// NeuroPLC — Auto-generated IEC 61131-3 SCL
// Graph: kan | Target: S71200Backend
// Work memory: 75KB | LUT points: 15
// Nodes: 11 | Ops: {'matmul': 3, 'standard_act': 2, 'bspline_lut': 2, 'add': 2, 'softmax': 1, 'argmax': 1}


DATA_BLOCK "NeuroPLC_Weights"
{ S7_Optimized_Access := 'FALSE' }
VERSION : 0.1
NON_RETAIN
   STRUCT

   // BsplineLUT 'l0_bspline': grid(15 pts) + table(16×28×15)
   w0 : ARRAY[0..14] OF REAL :=
[-3.0000000, -2.5714286, -2.1428571, -1.7142857, -1.2857143, -0.8571429, -0.4285714, 0.0
    0.4285714, 0.8571429, 1.2857143, 1.7142857, 2.1428571, 2.5714286, 3.0000000];
   w1 : ARRAY[0..6719] OF REAL :=
[-0.0537614, -0.0501507, -0.0466009, -0.0431086, -0.0396707, -0.0362841, -0.0329455, -0.0296518
    -0.0263998, -0.0231863, -0.0200081, -0.0168621, -0.0137450, -0.0106537, -0.0075850, 0.0036137
    0.0087966, 0.0140219, 0.0192753, 0.0245424, 0.0298091, 0.0350611, 0.0402840, 0.0454636
    0.0505857, 0.0556359, 0.0606001, 0.0654638, 0.0702129, 0.0748330, 0.0177914, 0.0204340
    0.0230393, 0.0256087, 0.0281433, 0.0306442, 0.0331128, 0.0355502, 0.0379576, 0.0403361
    0.0426870, 0.0450116, 0.0473109, 0.0495862, 0.0518386, 0.0911694, 0.0932300, 0.0951918
    0.0970447, 0.0987788, 0.1003839, 0.1018500, 0.1031669, 0.1043247, 0.1053133, 0.1061226
    0.1067426, 0.1071632, 0.1073743, 0.1073658, 0.1621530, 0.1624265, 0.1625151, 0.1624206
    0.1621450, 0.1616900, 0.1610576, 0.1602496, 0.1592678, 0.1581141, 0.1567904, 0.1552985
    0.1536403, 0.1518177, 0.1498324, 0.0235894, 0.0199670, 0.0162926, 0.0125813, 0.0088480
    0.0051075, 0.0013748, -0.0023352, -0.0060075, -0.0096273, -0.0131797, -0.0166496, -0.0200223
    -0.0232827, -0.0264160, 0.0037645, 0.0049106, 0.0061689, 0.0075391, 0.0090207, 0.0106134
    0.0123167, 0.0141303, 0.0160538, 0.0180869, 0.0202291, 0.0224800, 0.0248393, 0.0273066
    0.0298814, 0.1595527, 0.1622552, 0.1649406, 0.1675934, 0.1701985, 0.1727402, 0.1752033
    0.1775724, 0.1798320, 0.1819669, 0.1839615, 0.1858006, 0.1874687, 0.1889505, 0.1902305
    0.0697959, 0.0692244, 0.0685901, 0.0679135, 0.0672150, 0.0665149, 0.0658336, 0.0651916
    0.0646091, 0.0641067, 0.0637047, 0.0634234, 0.0632833, 0.0633048, 0.0635083, 0.0889156
    0.0916844, 0.0943388, 0.0968816, 0.0993158, 0.1016441, 0.1038697, 0.1059952, 0.1080237
    0.1099581, 0.1118012, 0.1135559, 0.1152252, 0.1168119, 0.1183189, -0.0411367, -0.0345732
    -0.0279382, -0.0212556, -0.0145492, -0.0078430, -0.0011607, 0.0054737, 0.0120364, 0.0185035
    0.0248511, 0.0310554, 0.0370926, 0.0429386, 0.0485698, 0.1426231, 0.1415560, 0.1405476
    0.1395973, 0.1387044, 0.1378686, 0.1370891, 0.1363655, 0.1356970, 0.1350832, 0.1345235
    0.1340173, 0.1335640, 0.1331631, 0.1328139, 0.2510517, 0.2566622, 0.2620918, 0.2673131
    0.2722991, 0.2770230, 0.2814575, 0.2855757, 0.2893504, 0.2927547, 0.2957615, 0.2983437
    0.3004743, 0.3021264, 0.3032727, 0.0229299, 0.0200585, 0.0170953, 0.0140589, 0.0109677
    0.0078400, 0.0046945, 0.0015496, -0.0015764, -0.0046649, -0.0076974, -0.0106555, -0.0135208
    -0.0162748, -0.0188990, 0.0368656, 0.0374461, 0.0380069, 0.0385353, 0.0390182, 0.0394428
    0.0397962, 0.0400654, 0.0402376, 0.0402999, 0.0402393, 0.0400429, 0.0396979, 0.0391914
    0.0385103, 0.2372042, 0.2373395, 0.2373046, 0.2371029, 0.2367378, 0.2362127, 0.2355310
    0.2346960, 0.2337111, 0.2325798, 0.2313054, 0.2298912, 0.2283408, 0.2266575, 0.2248445
    0.1274217, 0.1323916, 0.1373182, 0.1421699, 0.1469152, 0.1515225, 0.1559602, 0.1601968
    0.1642006, 0.1679402, 0.1713839, 0.1745002, 0.1772575, 0.1796242, 0.1815687, 0.0097799
    0.0143171, 0.0189285, 0.0236177, 0.0283886, 0.0332447, 0.0381899, 0.0432280, 0.0483625
    0.0535974, 0.0589362, 0.0643828, 0.0699409, 0.0756142, 0.0814065, 0.0746824, 0.0808143
    0.0870039, 0.0932227, 0.0994422, 0.1056337, 0.1117689, 0.1178190, 0.1237556, 0.1295501
    0.1351739, 0.1405987, 0.1457956, 0.1507363, 0.1553921, 0.1577364, 0.1559705, 0.1542206
    0.1524857, 0.1507643, 0.1490552, 0.1473571, 0.1456687, 0.1439888, 0.1423160, 0.1406490
    0.1389866, 0.1373274, 0.1356702, 0.1340137, 0.0440495, 0.0446013, 0.0452923, 0.0461173
    0.0470712, 0.0481487, 0.0493447, 0.0506540, 0.0520714, 0.0535917, 0.0552098, 0.0569205
    0.0587186, 0.0605990, 0.0625563, 0.1515065, 0.1420245, 0.1325012, 0.1229551, 0.1134045
    0.1038679, 0.0943635, 0.0849099, 0.0755254, 0.0662283, 0.0570372, 0.0479702, 0.0390460
    0.0302827, 0.0216989, 0.2110309, 0.2063019, 0.2015673, 0.1968229, 0.1920643, 0.1872871
    0.1824870, 0.1776595, 0.1728004, 0.1679052, 0.1629696, 0.1579892, 0.1529597, 0.1478766
    0.1427357, 0.1167147, 0.1155411, 0.1143786, 0.1132194, 0.1120559, 0.1108802, 0.1096847
    0.1084617, 0.1072033, 0.1059019, 0.1045497, 0.1031391, 0.1016622, 0.1001114, 0.0984789
    0.0612643, 0.0576810, 0.0542433, 0.0509556, 0.0478225, 0.0448487, 0.0420387, 0.0393971
    0.0369285, 0.0346374, 0.0325284, 0.0306060, 0.0288750, 0.0273397, 0.0260049, 0.0478268
    0.0498810, 0.0521120, 0.0545034, 0.0570387, 0.0597016, 0.0624757, 0.0653444, 0.0682915
    0.0713005, 0.0743550, 0.0774385, 0.0805347, 0.0836271, 0.0866994, 0.1196649, 0.1201896
    0.1209498, 0.1219383, 0.1231481, 0.1245723, 0.1262036, 0.1280351, 0.1300597, 0.1322704
    0.1346600, 0.1372216, 0.1399481, 0.1428323, 0.1458673, 0.1314654, 0.1267358, 0.1220911
    0.1175243, 0.1130283, 0.1085961, 0.1042207, 0.0998949, 0.0956117, 0.0913640, 0.0871449
    0.0829471, 0.0787638, 0.0745878, 0.0704120, 0.1482306, 0.1482909, 0.1482174, 0.1480233
    0.1477216, 0.1473256, 0.1468484, 0.1463031, 0.1457029, 0.1450608, 0.1443900, 0.1437037
    0.1430150, 0.1423371, 0.1416830, 0.0909267, 0.0942033, 0.0974144, 0.1005591, 0.1036367
    0.1066464, 0.1095874, 0.1124590, 0.1152604, 0.1179907, 0.1206493, 0.1232354, 0.1257481
    0.1281867, 0.1305504, 0.0411825, 0.0473991, 0.0535137, 0.0595173, 0.0654007, 0.0711547
    0.0767702, 0.0822381, 0.0875490, 0.0926940, 0.0976638, 0.1024494, 0.1070414, 0.1114309
    0.1156085, -0.1064937, -0.1066310, -0.1065970, -0.1063968, -0.1060358, -0.1055195, -0.1048531
    -0.1040420, -0.1030916, -0.1020073, -0.1007942, -0.0994579, -0.0980037, -0.0964369, -0.0947629
    0.1427321, 0.1493539, 0.1559923, 0.1626289, 0.1692458, 0.1758247, 0.1823476, 0.1887961
    0.1951523, 0.2013978, 0.2075146, 0.2134846, 0.2192896, 0.2249114, 0.2303318, 0.0604217
    0.0622943, 0.0641302, 0.0659233, 0.0676677, 0.0693572, 0.0709857, 0.0725473, 0.0740358
    0.0754452, 0.0767694, 0.0780024, 0.0791381, 0.0801705, 0.0810934, 0.1634620, 0.1628231
    0.1620056, 0.1610041, 0.1598133, 0.1584279, 0.1568425, 0.1550518, 0.1530505, 0.1508332
    0.1483946, 0.1457293, 0.1428322, 0.1396977, 0.1363206, 0.0563154, 0.0518884, 0.0473023
    0.0425774, 0.0377339, 0.0327920, 0.0277721, 0.0226943, 0.0175790, 0.0124463, 0.0073165
    0.0022098, -0.0028535, -0.0078531, -0.0127688, 0.0945771, 0.0939802, 0.0934194, 0.0929126
    0.0924782, 0.0921343, 0.0918991, 0.0917908, 0.0918276, 0.0920277, 0.0924092, 0.0929903
    0.0937893, 0.0948243, 0.0961135, 0.1597103, 0.1591299, 0.1584730, 0.1577443, 0.1569484
    0.1560901, 0.1551740, 0.1542049, 0.1531873, 0.1521261, 0.1510259, 0.1498914, 0.1487273
    0.1475383, 0.1463290, 0.1615033, 0.1660341, 0.1703599, 0.1744726, 0.1783642, 0.1820267
    0.1854521, 0.1886325, 0.1915598, 0.1942261, 0.1966232, 0.1987434, 0.2005784, 0.2021204
    0.2033613, 0.0735570, 0.0658352, 0.0581088, 0.0503981, 0.0427235, 0.0351053, 0.0275639
    0.0201196, 0.0127927, 0.0056037, -0.0014271, -0.0082794, -0.0149328, -0.0213670, -0.0275615
    0.1822264, 0.1774475, 0.1726047, 0.1676911, 0.1626996, 0.1576232, 0.1524548, 0.1471874
    0.1418141, 0.1363277, 0.1307212, 0.1249876, 0.1191199, 0.1131109, 0.1069538, 0.1921862
    0.1893261, 0.1864184, 0.1834680, 0.1804803, 0.1774603, 0.1744133, 0.1713443, 0.1682584
    0.1651610, 0.1620570, 0.1589516, 0.1558501, 0.1527575, 0.1496790, -0.0632336, -0.0648101
    -0.0662504, -0.0675372, -0.0686534, -0.0695816, -0.0703045, -0.0708049, -0.0710656, -0.0710692
    -0.0707984, -0.0702362, -0.0693650, -0.0681678, -0.0666272, 0.1172287, 0.1131316, 0.1088304
    0.1043208, 0.0995984, 0.0946590, 0.0894981, 0.0841114, 0.0784947, 0.0726435, 0.0665536
    0.0602206, 0.0536403, 0.0468081, 0.0397199, 0.1591443, 0.1524481, 0.1457851, 0.1391899
    0.1326966, 0.1263399, 0.1201540, 0.1141734, 0.1084325, 0.1029658, 0.0978075, 0.0929922
    0.0885542, 0.0845280, 0.0809479, -0.0802141, -0.0751070, -0.0699127, -0.0646468, -0.0593249
    -0.0539626, -0.0485752, -0.0431786, -0.0377880, -0.0324192, -0.0270877, -0.0218090, -0.0165986
    -0.0114722, -0.0064453, 0.0824098, 0.0763993, 0.0705333, 0.0648235, 0.0592816, 0.0539193
    0.0487485, 0.0437808, 0.0390279, 0.0345016, 0.0302137, 0.0261759, 0.0223999, 0.0188974
    0.0156802, 0.1799797, 0.1784663, 0.1767808, 0.1749217, 0.1728874, 0.1706764, 0.1682869
    0.1657176, 0.1629667, 0.1600327, 0.1569141, 0.1536092, 0.1501164, 0.1464343, 0.1425611
    -0.0496284, -0.0452828, -0.0409373, -0.0365933, -0.0322526, -0.0279167, -0.0235873, -0.0192659
    -0.0149543, -0.0106539, -0.0063663, -0.0020933, 0.0021636, 0.0064028, 0.0106226, 0.0450445
    0.0502692, 0.0554434, 0.0605487, 0.0655669, 0.0704798, 0.0752689, 0.0799160, 0.0844028
    0.0887111, 0.0928225, 0.0967188, 0.1003817, 0.1037928, 0.1069339, -0.0646169, -0.0560196
    -0.0472858, -0.0384308, -0.0294704, -0.0204202, -0.0112958, -0.0021127, 0.0071135, 0.0163671
    0.0256325, 0.0348942, 0.0441365, 0.0533439, 0.0625006, 0.0364423, 0.0390047, 0.0413258
    0.0434204, 0.0453037, 0.0469907, 0.0484963, 0.0498356, 0.0510236, 0.0520753, 0.0530057
    0.0538298, 0.0545627, 0.0552193, 0.0558146, 0.1494066, 0.1454436, 0.1415708, 0.1377844
    0.1340804, 0.1304549, 0.1269041, 0.1234239, 0.1200105, 0.1166601, 0.1133685, 0.1101320
    0.1069467, 0.1038086, 0.1007139, -0.0151529, -0.0096418, -0.0041800, 0.0012205, 0.0065474
    0.0117887, 0.0169322, 0.0219657, 0.0268772, 0.0316544, 0.0362853, 0.0407577, 0.0450594
    0.0491783, 0.0531024, 0.0760455, 0.0828511, 0.0895923, 0.0962519, 0.1028127, 0.1092577
    0.1155697, 0.1217317, 0.1277264, 0.1335369, 0.1391458, 0.1445363, 0.1496910, 0.1545929
    0.1592250, -0.0199655, -0.0125562, -0.0050469, 0.0025438, 0.0101974, 0.0178952, 0.0256188
    0.0333496, 0.0410690, 0.0487583, 0.0563991, 0.0639728, 0.0714608, 0.0788445, 0.0861054
    -0.0196776, -0.0178736, -0.0159748, -0.0139721, -0.0118560, -0.0096175, -0.0072471, -0.0047358
    -0.0020741, 0.0007470, 0.0037369, 0.0069048, 0.0102600, 0.0138117, 0.0175692, 0.0124894
    0.0173022, 0.0219949, 0.0265723, 0.0310388, 0.0353992, 0.0396580, 0.0438199, 0.0478895
    0.0518714, 0.0557702, 0.0595906, 0.0633373, 0.0670147, 0.0706276, 0.0248611, 0.0284164
    0.0320837, 0.0358641, 0.0397584, 0.0437678, 0.0478931, 0.0521354, 0.0564957, 0.0609750
    0.0655743, 0.0702945, 0.0751367, 0.0801018, 0.0851909, 0.1490314, 0.1533812, 0.1576221
    0.1617333, 0.1656937, 0.1694824, 0.1730786, 0.1764612, 0.1796093, 0.1825020, 0.1851182
    0.1874372, 0.1894379, 0.1910994, 0.1924008, 0.0541098, 0.0578787, 0.0616169, 0.0652991
    0.0689002, 0.0723947, 0.0757576, 0.0789636, 0.0819875, 0.0848040, 0.0873880, 0.0897141
    0.0917573, 0.0934922, 0.0948936, 0.0617447, 0.0675283, 0.0733681, 0.0792395, 0.0851180
    0.0909790, 0.0967979, 0.1025502, 0.1082113, 0.1137566, 0.1191614, 0.1244014, 0.1294519
    0.1342882, 0.1388859, -0.0461591, -0.0453256, -0.0443076, -0.0431073, -0.0417270, -0.0401691
    -0.0384360, -0.0365298, -0.0344530, -0.0322079, -0.0297967, -0.0272219, -0.0244857, -0.0215905
    -0.0185385, 0.0292693, 0.0302004, 0.0311640, 0.0321651, 0.0332088, 0.0343000, 0.0354438
    0.0366453, 0.0379094, 0.0392413, 0.0406458, 0.0421281, 0.0436931, 0.0453460, 0.0470917
    0.1551978, 0.1594762, 0.1635234, 0.1673317, 0.1708932, 0.1742002, 0.1772451, 0.1800199
    0.1825169, 0.1847285, 0.1866468, 0.1882641, 0.1895726, 0.1905645, 0.1912322, -0.0022298
    0.0015482, 0.0054057, 0.0093347, 0.0133276, 0.0173766, 0.0214738, 0.0256116, 0.0297821
    0.0339775, 0.0381901, 0.0424120, 0.0466356, 0.0508530, 0.0550565, 0.0832689, 0.0901474
    0.0970738, 0.1040439, 0.1110534, 0.1180982, 0.1251741, 0.1322769, 0.1394024, 0.1465464
    0.1537047, 0.1608732, 0.1680476, 0.1752237, 0.1823975, 0.0709989, 0.0702285, 0.0696263
    0.0691951, 0.0689377, 0.0688570, 0.0689556, 0.0692364, 0.0697023, 0.0703559, 0.0712001
    0.0722376, 0.0734714, 0.0749041, 0.0765386, 0.0713218, 0.0738626, 0.0762200, 0.0783959
    0.0803921, 0.0822106, 0.0838531, 0.0853217, 0.0866181, 0.0877443, 0.0887021, 0.0894935
    0.0901202, 0.0905842, 0.0908874, 0.1406779, 0.1441289, 0.1474667, 0.1506924, 0.1538070
    0.1568115, 0.1597070, 0.1624945, 0.1651749, 0.1677495, 0.1702191, 0.1725848, 0.1748478
    0.1770088, 0.1790691, 0.0130739, 0.0090535, 0.0049917, 0.0009004, -0.0032088, -0.0073243
    -0.0114343, -0.0155273, -0.0195916, -0.0236154, -0.0275873, -0.0314954, -0.0353281, -0.0390738
    -0.0427207, 0.0809735, 0.0798324, 0.0785689, 0.0771792, 0.0756592, 0.0740052, 0.0722131
    0.0702792, 0.0681993, 0.0659697, 0.0635865, 0.0610456, 0.0583432, 0.0554754, 0.0524383
    0.1908756, 0.1884213, 0.1857675, 0.1829149, 0.1798646, 0.1766175, 0.1731745, 0.1695365
    0.1657044, 0.1616793, 0.1574618, 0.1530531, 0.1484540, 0.1436654, 0.1386883, -0.1181388
    -0.1128441, -0.1073974, -0.1018071, -0.0960813, -0.0902284, -0.0842566, -0.0781741, -0.0719893
    -0.0657102, -0.0593453, -0.0529027, -0.0463907, -0.0398176, -0.0331916, -0.0020498, 0.0079060
    0.0177509, 0.0274740, 0.0370644, 0.0465111, 0.0558031, 0.0649296, 0.0738794, 0.0826418
    0.0912057, 0.0995603, 0.1076945, 0.1155974, 0.1232580, -0.0007446, -0.0019150, -0.0031143
    -0.0043173, -0.0054990, -0.0066342, -0.0076977, -0.0086645, -0.0095093, -0.0102072, -0.0107328
    -0.0110612, -0.0111671, -0.0110255, -0.0106112, 0.1774268, 0.1753455, 0.1732356, 0.1710882
    0.1688946, 0.1666464, 0.1643346, 0.1619507, 0.1594860, 0.1569317, 0.1542792, 0.1515199
    0.1486450, 0.1456458, 0.1425137, 0.1379051, 0.1349382, 0.1318155, 0.1285463, 0.1251401
    0.1216064, 0.1179545, 0.1141940, 0.1103341, 0.1063845, 0.1023545, 0.0982536, 0.0940911
    0.0898766, 0.0856195, 0.0633166, 0.0493134, 0.0352768, 0.0212369, 0.0072238, -0.0067325
    -0.0206019, -0.0343543, -0.0479595, -0.0613876, -0.0746085, -0.0875920, -0.1003081, -0.1127267
    -0.1248178, 0.1183318, 0.1136023, 0.1089029, 0.1042314, 0.0995855, 0.0949629, 0.0903612
    0.0857784, 0.0812119, 0.0766596, 0.0721192, 0.0675883, 0.0630647, 0.0585461, 0.0540302
    0.1106823, 0.1041894, 0.0975902, 0.0909071, 0.0841626, 0.0773792, 0.0705792, 0.0637853
    0.0570198, 0.0503051, 0.0436638, 0.0371183, 0.0306911, 0.0244045, 0.0182812, 0.0562573
    0.0481918, 0.0400543, 0.0318683, 0.0236572, 0.0154445, 0.0072537, -0.0008917, -0.0089682
    -0.0169524, -0.0248208, -0.0325500, -0.0401163, -0.0474965, -0.0546669, 0.2219241, 0.2176533
    0.2134451, 0.2093052, 0.2052390, 0.2012524, 0.1973507, 0.1935398, 0.1898251, 0.1862123
    0.1827069, 0.1793146, 0.1760410, 0.1728917, 0.1698723, 0.3312375, 0.3261927, 0.3209868
    0.3156299, 0.3101325, 0.3045048, 0.2987574, 0.2929004, 0.2869442, 0.2808991, 0.2747756
    0.2685839, 0.2623343, 0.2560374, 0.2497033, 0.1718789, 0.1756587, 0.1793987, 0.1830900
    0.1867239, 0.1902918, 0.1937850, 0.1971947, 0.2005122, 0.2037288, 0.2068357, 0.2098243
    0.2126858, 0.2154116, 0.2179928, 0.1224311, 0.1282386, 0.1340468, 0.1398439, 0.1456182
    0.1513580, 0.1570517, 0.1626873, 0.1682533, 0.1737379, 0.1791293, 0.1844160, 0.1895860
    0.1946277, 0.1995294, 0.0492804, 0.0562029, 0.0630472, 0.0698060, 0.0764722, 0.0830386
    0.0894981, 0.0958434, 0.1020674, 0.1081630, 0.1141229, 0.1199399, 0.1256070, 0.1311170
    0.1364626, 0.1061752, 0.1096911, 0.1131474, 0.1165290, 0.1198208, 0.1230075, 0.1260742
    0.1290057, 0.1317867, 0.1344023, 0.1368373, 0.1390765, 0.1411048, 0.1429072, 0.1444684
    0.0055067, 0.0101075, 0.0148682, 0.0197738, 0.0248092, 0.0299594, 0.0352094, 0.0405440
    0.0459484, 0.0514074, 0.0569060, 0.0624292, 0.0679618, 0.0734890, 0.0789956, 0.2030336
    0.2064162, 0.2097383, 0.2129931, 0.2161737, 0.2192730, 0.2222843, 0.2252005, 0.2280147
    0.2307200, 0.2333094, 0.2357761, 0.2381131, 0.2403134, 0.2423701, 0.0904342, 0.0915991
    0.0928258, 0.0941062, 0.0954321, 0.0967953, 0.0981878, 0.0996012, 0.1010275, 0.1024584
    0.1038859, 0.1053016, 0.1066976, 0.1080655, 0.1093972, 0.1280624, 0.1273501, 0.1266980
    0.1261149, 0.1256098, 0.1251912, 0.1248681, 0.1246492, 0.1245433, 0.1245592, 0.1247057
    0.1249917, 0.1254258, 0.1260169, 0.1267738, 0.1299709, 0.1307576, 0.1315505, 0.1323500
    0.1331564, 0.1339704, 0.1347923, 0.1356225, 0.1364616, 0.1373100, 0.1381681, 0.1390364
    0.1399154, 0.1408054, 0.1417070, 0.1533135, 0.1507089, 0.1480348, 0.1452944, 0.1424904
    0.1396261, 0.1367043, 0.1337281, 0.1307005, 0.1276246, 0.1245032, 0.1213395, 0.1181364
    0.1148970, 0.1116242, 0.0754236, 0.0751954, 0.0749772, 0.0747602, 0.0745356, 0.0742946
    0.0740284, 0.0737282, 0.0733853, 0.0729909, 0.0725361, 0.0720122, 0.0714104, 0.0707219
    0.0699379, 0.2758769, 0.2724863, 0.2687611, 0.2647197, 0.2603807, 0.2557624, 0.2508835
    0.2457622, 0.2404172, 0.2348669, 0.2291298, 0.2232242, 0.2171688, 0.2109820, 0.2046822
    0.0770989, 0.0772505, 0.0775468, 0.0779858, 0.0785653, 0.0792835, 0.0801382, 0.0811273
    0.0822489, 0.0835009, 0.0848812, 0.0863879, 0.0880188, 0.0897719, 0.0916453, 0.1377456
    0.1380898, 0.1384590, 0.1388540, 0.1392763, 0.1397269, 0.1402069, 0.1407176, 0.1412600
    0.1418354, 0.1424448, 0.1430894, 0.1437705, 0.1444890, 0.1452463, 0.0905914, 0.0893503
    0.0881403, 0.0869641, 0.0858247, 0.0847249, 0.0836674, 0.0826551, 0.0816908, 0.0807774
    0.0799175, 0.0791142, 0.0783702, 0.0776883, 0.0770713, 0.0768078, 0.0747090, 0.0725560
    0.0703614, 0.0681377, 0.0658974, 0.0636532, 0.0614176, 0.0592031, 0.0570223, 0.0548878
    0.0528120, 0.0508076, 0.0488871, 0.0470630, 0.0018665, 0.0055140, 0.0092878, 0.0131758
    0.0171657, 0.0212453, 0.0254025, 0.0296251, 0.0339007, 0.0382174, 0.0425627, 0.0469246
    0.0512909, 0.0556493, 0.0599876, 0.1362334, 0.1320360, 0.1276240, 0.1230101, 0.1182072
    0.1132279, 0.1080852, 0.1027917, 0.0973602, 0.0918035, 0.0861343, 0.0803655, 0.0745097
    0.0685798, 0.0625885, 0.0739216, 0.0777187, 0.0816159, 0.0855995, 0.0896565, 0.0937732
    0.0979364, 0.1021327, 0.1063487, 0.1105710, 0.1147861, 0.1189809, 0.1231417, 0.1272554
    0.1313084, 0.1225641, 0.1228170, 0.1230709, 0.1233162, 0.1235429, 0.1237414, 0.1239020
    0.1240148, 0.1240701, 0.1240582, 0.1239692, 0.1237935, 0.1235212, 0.1231427, 0.1226481
    0.0764033, 0.0779041, 0.0794761, 0.0811008, 0.0827599, 0.0844351, 0.0861080, 0.0877602
    0.0893733, 0.0909290, 0.0924088, 0.0937945, 0.0950676, 0.0962098, 0.0972026, 0.1156939
    0.1193963, 0.1228430, 0.1260415, 0.1289993, 0.1317239, 0.1342227, 0.1365035, 0.1385735
    0.1404405, 0.1421117, 0.1435948, 0.1448973, 0.1460266, 0.1469904, 0.0673942, 0.0704027
    0.0733808, 0.0763299, 0.0792510, 0.0821455, 0.0850145, 0.0878592, 0.0906810, 0.0934810
    0.0962604, 0.0990204, 0.1017624, 0.1044874, 0.1071967, 0.0388152, 0.0469437, 0.0549675
    0.0628623, 0.0706043, 0.0781692, 0.0855331, 0.0926718, 0.0995613, 0.1061776, 0.1124965
    0.1184940, 0.1241459, 0.1294284, 0.1343171, 0.1772938, 0.1717090, 0.1661408, 0.1606062
    0.1551221, 0.1497055, 0.1443732, 0.1391423, 0.1340295, 0.1290519, 0.1242263, 0.1195697
    0.1150991, 0.1108312, 0.1067832, 0.1667371, 0.1745140, 0.1819698, 0.1890907, 0.1958626
    0.2022715, 0.2083035, 0.2139444, 0.2191803, 0.2239972, 0.2283811, 0.2323180, 0.2357939
    0.2387947, 0.2413065, 0.1465034, 0.1458727, 0.1451484, 0.1443270, 0.1434050, 0.1423789
    0.1412452, 0.1400004, 0.1386409, 0.1371633, 0.1355640, 0.1338395, 0.1319864, 0.1300010
    0.1278800, -0.1464676, -0.1331242, -0.1196480, -0.1060719, -0.0924292, -0.0787528, -0.0650760
    -0.0514318, -0.0378533, -0.0243737, -0.0110261, 0.0021565, 0.0151410, 0.0278942, 0.0403829
    0.0219379, 0.0184042, 0.0149580, 0.0116003, 0.0083324, 0.0051556, 0.0020711, -0.0009198
    -0.0038158, -0.0066158, -0.0093184, -0.0119225, -0.0144268, -0.0168299, -0.0191308, -0.0799424
    -0.0830510, -0.0860327, -0.0888876, -0.0916160, -0.0942182, -0.0966944, -0.0990448, -0.1012698
    -0.1033695, -0.1053442, -0.1071942, -0.1089198, -0.1105211, -0.1119984, 0.1063759, 0.1058369
    0.1052956, 0.1047466, 0.1041849, 0.1036053, 0.1030025, 0.1023714, 0.1017069, 0.1010037
    0.1002566, 0.0994605, 0.0986103, 0.0977007, 0.0967265, -0.0524474, -0.0499474, -0.0472491
    -0.0443565, -0.0412736, -0.0380045, -0.0345532, -0.0309238, -0.0271203, -0.0231467, -0.0190072
    -0.0147057, -0.0102462, -0.0056329, -0.0008698, -0.0401886, -0.0425021, -0.0449156, -0.0474036
    -0.0499410, -0.0525023, -0.0550621, -0.0575950, -0.0600758, -0.0624789, -0.0647791, -0.0669510
    -0.0689691, -0.0708082, -0.0724429, 0.0068997, 0.0025731, -0.0018010, -0.0061969, -0.0105893
    -0.0149526, -0.0192613, -0.0234899, -0.0276128, -0.0316047, -0.0354398, -0.0390929, -0.0425383
    -0.0457506, -0.0487042, 0.0460935, 0.0446672, 0.0431436, 0.0415249, 0.0398133, 0.0380112
    0.0361207, 0.0341442, 0.0320837, 0.0299417, 0.0277203, 0.0254217, 0.0230483, 0.0206022
    0.0180857, 0.0362551, 0.0359917, 0.0356584, 0.0352565, 0.0347877, 0.0342534, 0.0336551
    0.0329943, 0.0322726, 0.0314914, 0.0306522, 0.0297565, 0.0288058, 0.0278016, 0.0267454
    0.1229962, 0.1128694, 0.1027529, 0.0926827, 0.0826947, 0.0728249, 0.0631090, 0.0535829
    0.0442827, 0.0352441, 0.0265031, 0.0180955, 0.0100574, 0.0024244, -0.0047673, -0.0390921
    -0.0409484, -0.0426025, -0.0440575, -0.0453165, -0.0463824, -0.0472584, -0.0479475, -0.0484527
    -0.0487771, -0.0489238, -0.0488957, -0.0486959, -0.0483276, -0.0477937, 0.0402361, 0.0420451
    0.0438251, 0.0455756, 0.0472959, 0.0489854, 0.0506435, 0.0522696, 0.0538632, 0.0554235
    0.0569500, 0.0584422, 0.0598992, 0.0613207, 0.0627060, -0.0578378, -0.0600211, -0.0621784
    -0.0642941, -0.0663524, -0.0683375, -0.0702337, -0.0720250, -0.0736959, -0.0752304, -0.0766129
    -0.0778275, -0.0788584, -0.0796900, -0.0803063, -0.0276505, -0.0345807, -0.0413763, -0.0480331
    -0.0545471, -0.0609143, -0.0671306, -0.0731920, -0.0790944, -0.0848337, -0.0904060, -0.0958071
    -0.1010331, -0.1060798, -0.1109432, -0.0786863, -0.0790071, -0.0793080, -0.0795758, -0.0797971
    -0.0799585, -0.0800469, -0.0800488, -0.0799510, -0.0797402, -0.0794029, -0.0789260, -0.0782961
    -0.0774999, -0.0765241, 0.0213712, 0.0235205, 0.0256513, 0.0277667, 0.0298702, 0.0319649
    0.0340539, 0.0361407, 0.0382283, 0.0403200, 0.0424190, 0.0445287, 0.0466521, 0.0487925
    0.0509532, 0.0470440, 0.0409675, 0.0348353, 0.0286634, 0.0224677, 0.0162640, 0.0100684
    0.0038966, -0.0022354, -0.0083116, -0.0143163, -0.0202335, -0.0260472, -0.0317417, -0.0373009
    0.0554819, 0.0524533, 0.0493854, 0.0462786, 0.0431332, 0.0399497, 0.0367285, 0.0334701
    0.0301748, 0.0268430, 0.0234752, 0.0200718, 0.0166333, 0.0131599, 0.0096522, -0.0472854
    -0.0443733, -0.0413744, -0.0382941, -0.0351381, -0.0319120, -0.0286213, -0.0252716, -0.0218685
    -0.0184174, -0.0149240, -0.0113939, -0.0078326, -0.0042456, -0.0006386, 0.2066563, 0.1984604
    0.1899513, 0.1811467, 0.1720641, 0.1627212, 0.1531354, 0.1433243, 0.1333057, 0.1230969
    0.1127157, 0.1021795, 0.0915059, 0.0807126, 0.0698171, 0.2430425, 0.2368604, 0.2303846
    0.2236263, 0.2165967, 0.2093072, 0.2017691, 0.1939936, 0.1859921, 0.1777758, 0.1693560
    0.1607441, 0.1519513, 0.1429889, 0.1338682, -0.2294966, -0.2238292, -0.2179271, -0.2117862
    -0.2054024, -0.1987716, -0.1918898, -0.1847527, -0.1773564, -0.1696967, -0.1617694, -0.1535706
    -0.1450962, -0.1363419, -0.1273037, -0.0534835, -0.0518626, -0.0502081, -0.0485070, -0.0467464
    -0.0449133, -0.0429948, -0.0409777, -0.0388492, -0.0365964, -0.0342061, -0.0316654, -0.0289615
    -0.0260812, -0.0230116, -0.0738918, -0.0681270, -0.0624695, -0.0569120, -0.0514472, -0.0460679
    -0.0407668, -0.0355367, -0.0303702, -0.0252601, -0.0201992, -0.0151801, -0.0101956, -0.0052385
    -0.0003014, -0.1733572, -0.1706521, -0.1679701, -0.1652953, -0.1626123, -0.1599054, -0.1571589
    -0.1543573, -0.1514847, -0.1485257, -0.1454645, -0.1422856, -0.1389732, -0.1355117, -0.1318855
    -0.1211167, -0.1186958, -0.1162400, -0.1137493, -0.1112237, -0.1086634, -0.1060684, -0.1034386
    -0.1007743, -0.0980754, -0.0953419, -0.0925739, -0.0897715, -0.0869348, -0.0840637, -0.1646881
    -0.1559299, -0.1470360, -0.1380355, -0.1289572, -0.1198299, -0.1106827, -0.1015443, -0.0924438
    -0.0834100, -0.0744717, -0.0656579, -0.0569975, -0.0485193, -0.0402523, -0.0817973, -0.0730933
    -0.0642312, -0.0552295, -0.0461065, -0.0368805, -0.0275698, -0.0181927, -0.0087677, 0.0006871
    0.0101533, 0.0196125, 0.0290465, 0.0384369, 0.0477654, 0.0163655, 0.0131517, 0.0101446
    0.0073348, 0.0047129, 0.0022695, -0.0000050, -0.0021197, -0.0040842, -0.0059079, -0.0076002
    -0.0091705, -0.0106281, -0.0119826, -0.0132432, 0.1066189, 0.1081075, 0.1096451, 0.1112214
    0.1128261, 0.1144488, 0.1160794, 0.1177076, 0.1193229, 0.1209153, 0.1224743, 0.1239896
    0.1254511, 0.1268484, 0.1281711, 0.1267634, 0.1300867, 0.1334209, 0.1367561, 0.1400827
    0.1433908, 0.1466706, 0.1499123, 0.1531061, 0.1562422, 0.1593107, 0.1623020, 0.1652061
    0.1680134, 0.1707140, 0.1024532, 0.1037427, 0.1049064, 0.1059469, 0.1068673, 0.1076704
    0.1083589, 0.1089356, 0.1094036, 0.1097654, 0.1100241, 0.1101824, 0.1102432, 0.1102092
    0.1100834, 0.0440706, 0.0458766, 0.0476553, 0.0494080, 0.0511363, 0.0528416, 0.0545253
    0.0561887, 0.0578334, 0.0594607, 0.0610720, 0.0626688, 0.0642525, 0.0658246, 0.0673864
    -0.0485841, -0.0409054, -0.0330825, -0.0251116, -0.0169887, -0.0087100, -0.0002714, 0.0083308
    0.0171006, 0.0260419, 0.0351585, 0.0444545, 0.0539337, 0.0636000, 0.0734574, 0.1719400
    0.1734631, 0.1749307, 0.1763346, 0.1776664, 0.1789180, 0.1800810, 0.1811472, 0.1821083
    0.1829559, 0.1836818, 0.1842779, 0.1847356, 0.1850469, 0.1852033, 0.0836945, 0.0829144
    0.0820091, 0.0809680, 0.0797808, 0.0784369, 0.0769259, 0.0752372, 0.0733605, 0.0712852
    0.0690009, 0.0664970, 0.0637631, 0.0607888, 0.0575636, 0.0451547, 0.0443564, 0.0433699
    0.0422019, 0.0408591, 0.0393482, 0.0376759, 0.0358490, 0.0338742, 0.0317582, 0.0295077
    0.0271295, 0.0246304, 0.0220170, 0.0192960, 0.1446830, 0.1442651, 0.1438369, 0.1434112
    0.1430013, 0.1426201, 0.1422805, 0.1419956, 0.1417785, 0.1416420, 0.1415993, 0.1416632
    0.1418470, 0.1421634, 0.1426256, -0.0780212, -0.0782113, -0.0783461, -0.0784252, -0.0784484
    -0.0784154, -0.0783258, -0.0781794, -0.0779759, -0.0777149, -0.0773962, -0.0770194, -0.0765842
    -0.0760904, -0.0755376, 0.2056785, 0.2034542, 0.2009305, 0.1981261, 0.1950600, 0.1917508
    0.1882173, 0.1844784, 0.1805528, 0.1764593, 0.1722167, 0.1678438, 0.1633593, 0.1587822
    0.1541310, 0.1056817, 0.0955098, 0.0850380, 0.0743014, 0.0633348, 0.0521733, 0.0408519
    0.0294056, 0.0178693, 0.0062781, -0.0053330, -0.0169291, -0.0284751, -0.0399361, -0.0512770
    0.0299433, 0.0223843, 0.0149406, 0.0076058, 0.0003734, -0.0067630, -0.0138100, -0.0207740
    -0.0276615, -0.0344789, -0.0412327, -0.0479294, -0.0545755, -0.0611774, -0.0677417, 0.1432800
    0.1365236, 0.1298036, 0.1231296, 0.1165111, 0.1099579, 0.1034795, 0.0970856, 0.0907857
    0.0845895, 0.0785066, 0.0725466, 0.0667192, 0.0610339, 0.0555004, -0.0302912, -0.0280554
    -0.0257948, -0.0235061, -0.0211860, -0.0188312, -0.0164385, -0.0140044, -0.0115256, -0.0089990
    -0.0064211, -0.0037886, -0.0010983, 0.0016532, 0.0044692, 0.1403525, 0.1435867, 0.1466069
    0.1493943, 0.1519307, 0.1541973, 0.1561757, 0.1578473, 0.1591936, 0.1601962, 0.1608364
    0.1610958, 0.1609558, 0.1603979, 0.1594036, -0.0224080, -0.0231706, -0.0235986, -0.0236903
    -0.0234441, -0.0228584, -0.0219317, -0.0206623, -0.0190486, -0.0170891, -0.0147821, -0.0121260
    -0.0091192, -0.0057602, -0.0020472, 0.0048894, 0.0037833, 0.0026298, 0.0014329, 0.0001967
    -0.0010748, -0.0023775, -0.0037073, -0.0050602, -0.0064321, -0.0078189, -0.0092166, -0.0106211
    -0.0120284, -0.0134344, 0.1748016, 0.1674656, 0.1599554, 0.1522917, 0.1444954, 0.1365874
    0.1285885, 0.1205195, 0.1124012, 0.1042545, 0.0961002, 0.0879591, 0.0798522, 0.0718001
    0.0638238, 0.2813404, 0.2743131, 0.2670321, 0.2595086, 0.2517535, 0.2437782, 0.2355935
    0.2272108, 0.2186410, 0.2098953, 0.2009848, 0.1919205, 0.1827137, 0.1733754, 0.1639168
    -0.1227151, -0.1167440, -0.1105694, -0.1042075, -0.0976747, -0.0909872, -0.0841613, -0.0772134
    -0.0701597, -0.0630166, -0.0558003, -0.0485272, -0.0412136, -0.0338758, -0.0265300, 0.0716502
    0.0740325, 0.0763472, 0.0785967, 0.0807833, 0.0829093, 0.0849771, 0.0869889, 0.0889471
    0.0908540, 0.0927120, 0.0945233, 0.0962903, 0.0980153, 0.0997006, 0.1102683, 0.1225627
    0.1347638, 0.1468584, 0.1588335, 0.1706758, 0.1823722, 0.1939096, 0.2052749, 0.2164549
    0.2274364, 0.2382064, 0.2487517, 0.2590591, 0.2691154, 0.2098262, 0.2144697, 0.2187104
    0.2225624, 0.2260398, 0.2291567, 0.2319272, 0.2343654, 0.2364854, 0.2383013, 0.2398272
    0.2410773, 0.2420656, 0.2428063, 0.2433134, 0.1236384, 0.1234346, 0.1231693, 0.1228465
    0.1224701, 0.1220440, 0.1215722, 0.1210586, 0.1205071, 0.1199218, 0.1193064, 0.1186650
    0.1180016, 0.1173200, 0.1166241, -0.0358423, -0.0302241, -0.0246765, -0.0192003, -0.0137963
    -0.0084654, -0.0032083, 0.0019742, 0.0070812, 0.0121121, 0.0170660, 0.0219421, 0.0267396
    0.0314578, 0.0360958, -0.0184696, -0.0128896, -0.0074545, -0.0021679, 0.0029665, 0.0079452
    0.0127643, 0.0174204, 0.0219097, 0.0262287, 0.0303736, 0.0343408, 0.0381267, 0.0417277
    0.0451400, -0.1589818, -0.1530462, -0.1471289, -0.1412169, -0.1352974, -0.1293573, -0.1233838
    -0.1173639, -0.1112847, -0.1051332, -0.0988965, -0.0925616, -0.0861157, -0.0795457, -0.0728388
    -0.0915808, -0.0858980, -0.0802137, -0.0745331, -0.0688611, -0.0632027, -0.0575628, -0.0519466
    -0.0463591, -0.0408051, -0.0352897, -0.0298179, -0.0243948, -0.0190252, -0.0137143, -0.0835398
    -0.0728436, -0.0621097, -0.0513475, -0.0405668, -0.0297773, -0.0189886, -0.0082104, 0.0025477
    0.0132760, 0.0239648, 0.0346044, 0.0451853, 0.0556977, 0.0661319, -0.0592816, -0.0595268
    -0.0600139, -0.0607121, -0.0615909, -0.0626199, -0.0637683, -0.0650056, -0.0663012, -0.0676246
    -0.0689452, -0.0702323, -0.0714555, -0.0725841, -0.0735876, 0.0978256, 0.0979407, 0.0979876
    0.0979614, 0.0978575, 0.0976711, 0.0973975, 0.0970319, 0.0965695, 0.0960057, 0.0953356
    0.0945545, 0.0936577, 0.0926404, 0.0914979, -0.1088112, -0.1062184, -0.1035894, -0.1009293
    -0.0982433, -0.0955364, -0.0928137, -0.0900805, -0.0873417, -0.0846026, -0.0818682, -0.0791436
    -0.0764340, -0.0737444, -0.0710801, 0.0581553, 0.0553071, 0.0523084, 0.0491769, 0.0459304
    0.0425867, 0.0391635, 0.0356786, 0.0321498, 0.0285947, 0.0250312, 0.0214770, 0.0179500
    0.0144677, 0.0110481, -0.0312003, -0.0265061, -0.0215812, -0.0164328, -0.0110683, -0.0054952
    0.0002792, 0.0062476, 0.0124024, 0.0187363, 0.0252420, 0.0319121, 0.0387391, 0.0457157
    0.0528345, 0.0662310, 0.0672577, 0.0681709, 0.0689749, 0.0696742, 0.0702732, 0.0707762
    0.0711877, 0.0715121, 0.0717537, 0.0719170, 0.0720064, 0.0720262, 0.0719809, 0.0718749
    -0.0591723, -0.0535568, -0.0479641, -0.0424035, -0.0368841, -0.0314154, -0.0260063, -0.0206662
    -0.0154042, -0.0102296, -0.0051516, -0.0001794, 0.0046778, 0.0094108, 0.0140103, 0.1534036
    0.1555018, 0.1573710, 0.1590074, 0.1604071, 0.1615662, 0.1624808, 0.1631471, 0.1635612
    0.1637191, 0.1636170, 0.1632512, 0.1626176, 0.1617124, 0.1605317, -0.0163877, -0.0142709
    -0.0121985, -0.0101703, -0.0081860, -0.0062452, -0.0043479, -0.0024936, -0.0006821, 0.0010869
    0.0028135, 0.0044981, 0.0061410, 0.0077424, 0.0093026, 0.1683819, 0.1601295, 0.1516897
    0.1430965, 0.1343842, 0.1255870, 0.1167388, 0.1078739, 0.0990264, 0.0902305, 0.0815202
    0.0729298, 0.0644934, 0.0562450, 0.0482189, 0.0277282, 0.0297071, 0.0315788, 0.0333443
    0.0350050, 0.0365621, 0.0380169, 0.0393705, 0.0406241, 0.0417791, 0.0428366, 0.0437978
    0.0446641, 0.0454366, 0.0461166, 0.0431365, 0.0400386, 0.0370491, 0.0341767, 0.0314303
    0.0288187, 0.0263508, 0.0240353, 0.0218811, 0.0198970, 0.0180919, 0.0164745, 0.0150537
    0.0138383, 0.0128371, -0.0379476, -0.0376845, -0.0374638, -0.0372767, -0.0371142, -0.0369676
    -0.0368279, -0.0366863, -0.0365340, -0.0363621, -0.0361617, -0.0359240, -0.0356401, -0.0353011
    -0.0348983, 0.1160417, 0.1164429, 0.1166190, 0.1165743, 0.1163133, 0.1158405, 0.1151602
    0.1142770, 0.1131953, 0.1119195, 0.1104540, 0.1088034, 0.1069720, 0.1049642, 0.1027846
    -0.0046175, -0.0061991, -0.0076816, -0.0090646, -0.0103474, -0.0115296, -0.0126105, -0.0135896
    -0.0144664, -0.0152402, -0.0159105, -0.0164768, -0.0169384, -0.0172949, -0.0175456, 0.0451990
    0.0463734, 0.0473254, 0.0480687, 0.0486170, 0.0489840, 0.0491835, 0.0492290, 0.0491343
    0.0489131, 0.0485790, 0.0481459, 0.0476272, 0.0470369, 0.0463885, -0.1264566, -0.1190462
    -0.1114213, -0.1035908, -0.0955636, -0.0873487, -0.0789551, -0.0703916, -0.0616672, -0.0527909
    -0.0437716, -0.0346182, -0.0253396, -0.0159449, -0.0064429, 0.0945059, 0.0949724, 0.0954826
    0.0960497, 0.0966864, 0.0974060, 0.0982213, 0.0991454, 0.1001913, 0.1013720, 0.1027005
    0.1041898, 0.1058530, 0.1077029, 0.1097527, 0.0188506, 0.0162768, 0.0138876, 0.0116817
    0.0096579, 0.0078151, 0.0061521, 0.0046676, 0.0033605, 0.0022296, 0.0012736, 0.0004915
    -0.0001181, -0.0005562, -0.0008242, 0.0972443, 0.0940955, 0.0906709, 0.0869859, 0.0830556
    0.0788956, 0.0745210, 0.0699473, 0.0651896, 0.0602634, 0.0551839, 0.0499665, 0.0446265
    0.0391791, 0.0336398, 0.2299667, 0.2236568, 0.2170815, 0.2102544, 0.2031892, 0.1958997
    0.1883994, 0.1807021, 0.1728216, 0.1647715, 0.1565654, 0.1482172, 0.1397404, 0.1311487
    0.1224560, 0.1817064, 0.1786804, 0.1755636, 0.1723513, 0.1690391, 0.1656223, 0.1620962
    0.1584563, 0.1546980, 0.1508167, 0.1468077, 0.1426665, 0.1383885, 0.1339690, 0.1294035
    0.2677977, 0.2624427, 0.2569969, 0.2514781, 0.2459046, 0.2402945, 0.2346660, 0.2290372
    0.2234263, 0.2178514, 0.2123306, 0.2068821, 0.2015240, 0.1962745, 0.1911516, 0.2378129
    0.2257855, 0.2135410, 0.2011079, 0.1885143, 0.1757886, 0.1629592, 0.1500544, 0.1371024
    0.1241316, 0.1111703, 0.0982467, 0.0853894, 0.0726264, 0.0599862, 0.1316196, 0.1299897
    0.1284343, 0.1269458, 0.1255164, 0.1241385, 0.1228041, 0.1215057, 0.1202354, 0.1189855
    0.1177484, 0.1165162, 0.1152812, 0.1140357, 0.1127719, 0.0035808, 0.0141847, 0.0245993
    0.0348300, 0.0448826, 0.0547627, 0.0644760, 0.0740281, 0.0834246, 0.0926713, 0.1017736
    0.1107373, 0.1195681, 0.1282716, 0.1368533, 0.1038344, 0.1049576, 0.1060819, 0.1072011
    0.1083094, 0.1094007, 0.1104691, 0.1115086, 0.1125133, 0.1134771, 0.1143940, 0.1152582
    0.1160636, 0.1168043, 0.1174742, 0.1234559, 0.1209693, 0.1185037, 0.1160651, 0.1136594
    0.1112923, 0.1089697, 0.1066975, 0.1044815, 0.1023275, 0.1002415, 0.0982292, 0.0962965
    0.0944492, 0.0926933, -0.0080725, -0.0115148, -0.0148939, -0.0181990, -0.0214192, -0.0245438
    -0.0275620, -0.0304630, -0.0332361, -0.0358703, -0.0383549, -0.0406792, -0.0428324, -0.0448036
    -0.0465820, 0.0786227, 0.0774376, 0.0762180, 0.0749648, 0.0736790, 0.0723614, 0.0710129
    0.0696344, 0.0682269, 0.0667912, 0.0653283, 0.0638390, 0.0623243, 0.0607851, 0.0592223
    0.2340910, 0.2339238, 0.2334136, 0.2325522, 0.2313318, 0.2297445, 0.2277821, 0.2254369
    0.2227008, 0.2195658, 0.2160240, 0.2120674, 0.2076881, 0.2028781, 0.1976294, 0.0918500
    0.0925124, 0.0931616, 0.0937999, 0.0944295, 0.0950527, 0.0956717, 0.0962887, 0.0969060
    0.0975258, 0.0981503, 0.0987817, 0.0994224, 0.1000746, 0.1007404, 0.0606257, 0.0586222
    0.0567502, 0.0550141, 0.0534181, 0.0519667, 0.0506642, 0.0495149, 0.0485233, 0.0476937
    0.0470303, 0.0465377, 0.0462201, 0.0460819, 0.0461274, 0.1334510, 0.1322172, 0.1308804
    0.1294602, 0.1279766, 0.1264494, 0.1248983, 0.1233431, 0.1218037, 0.1202999, 0.1188515
    0.1174783, 0.1162001, 0.1150367, 0.1140079, 0.0197822, 0.0186880, 0.0175480, 0.0163653
    0.0151425, 0.0138827, 0.0125888, 0.0112635, 0.0099098, 0.0085306, 0.0071287, 0.0057072
    0.0042687, 0.0028163, 0.0013528, 0.0031245, 0.0026402, 0.0022171, 0.0018585, 0.0015677
    0.0013479, 0.0012022, 0.0011341, 0.0011466, 0.0012430, 0.0014267, 0.0017008, 0.0020685
    0.0025332, 0.0030980, 0.0377714, 0.0419777, 0.0463990, 0.0510148, 0.0558049, 0.0607489
    0.0658267, 0.0710178, 0.0763019, 0.0816588, 0.0870681, 0.0925096, 0.0979630, 0.1034078
    0.1088239, 0.1375776, 0.1375575, 0.1373740, 0.1370368, 0.1365557, 0.1359406, 0.1352013
    0.1343476, 0.1333894, 0.1323365, 0.1311986, 0.1299857, 0.1287075, 0.1273740, 0.1259948
    -0.1421038, -0.1365574, -0.1308133, -0.1248704, -0.1187279, -0.1123849, -0.1058404, -0.0990935
    -0.0921432, -0.0849887, -0.0776290, -0.0700631, -0.0622902, -0.0543093, -0.0461195, 0.0839307
    0.0920187, 0.1000085, 0.1078828, 0.1156247, 0.1232170, 0.1306426, 0.1378844, 0.1449253
    0.1517483, 0.1583360, 0.1646716, 0.1707378, 0.1765176, 0.1819938, 0.1568167, 0.1555951
    0.1541871, 0.1525968, 0.1508281, 0.1488851, 0.1467720, 0.1444927, 0.1420514, 0.1394521
    0.1366988, 0.1337956, 0.1307466, 0.1275558, 0.1242273, -0.0819356, -0.0749619, -0.0679275
    -0.0608395, -0.0537054, -0.0465324, -0.0393277, -0.0320986, -0.0248525, -0.0175966, -0.0103381
    -0.0030845, 0.0041572, 0.0113795, 0.0185752, 0.1820766, 0.1847949, 0.1872098, 0.1893105
    0.1910861, 0.1925258, 0.1936189, 0.1943544, 0.1947216, 0.1947095, 0.1943074, 0.1935045
    0.1922899, 0.1906527, 0.1885822, -0.0076931, -0.0099297, -0.0122230, -0.0145557, -0.0169104
    -0.0192699, -0.0216168, -0.0239338, -0.0262036, -0.0284088, -0.0305323, -0.0325566, -0.0344644
    -0.0362384, -0.0378614, 0.0374423, 0.0409134, 0.0444555, 0.0480605, 0.0517197, 0.0554249
    0.0591676, 0.0629394, 0.0667319, 0.0705367, 0.0743453, 0.0781495, 0.0819407, 0.0857107
    0.0894508, -0.0477527, -0.0446793, -0.0414355, -0.0380280, -0.0344633, -0.0307480, -0.0268889
    -0.0228923, -0.0187651, -0.0145137, -0.0101447, -0.0056649, -0.0010807, 0.0036012, 0.0083742
    0.0452007, 0.0379412, 0.0306638, 0.0233807, 0.0161044, 0.0088471, 0.0016212, -0.0055610
    -0.0126872, -0.0197451, -0.0267222, -0.0336064, -0.0403853, -0.0470465, -0.0535777, 0.0340680
    0.0324948, 0.0308646, 0.0292006, 0.0275258, 0.0258635, 0.0242368, 0.0226690, 0.0211832
    0.0198026, 0.0185503, 0.0174496, 0.0165236, 0.0157955, 0.0152884, 0.1499726, 0.1445799
    0.1393008, 0.1341326, 0.1290728, 0.1241187, 0.1192677, 0.1145172, 0.1098646, 0.1053073
    0.1008426, 0.0964679, 0.0921807, 0.0879783, 0.0838581, -0.1363414, -0.1354629, -0.1341214
    -0.1323354, -0.1301234, -0.1275037, -0.1244950, -0.1211155, -0.1173838, -0.1133184, -0.1089376
    -0.1042600, -0.0993040, -0.0940881, -0.0886307, 0.1193212, 0.1198225, 0.1202924, 0.1207296
    0.1211325, 0.1214999, 0.1218301, 0.1221219, 0.1223738, 0.1225843, 0.1227520, 0.1228755
    0.1229533, 0.1229841, 0.1229664, 0.0643094, 0.0664000, 0.0686213, 0.0709584, 0.0733966
    0.0759210, 0.0785170, 0.0811698, 0.0838645, 0.0865864, 0.0893207, 0.0920527, 0.0947675
    0.0974504, 0.1000866, 0.0684055, 0.0626766, 0.0569658, 0.0512835, 0.0456401, 0.0400461
    0.0345119, 0.0290481, 0.0236649, 0.0183730, 0.0131827, 0.0081044, 0.0031487, -0.0016741
    -0.0063534, 0.0475031, 0.0364922, 0.0253569, 0.0141221, 0.0028128, -0.0085461, -0.0199297
    -0.0313130, -0.0426711, -0.0539791, -0.0652119, -0.0763448, -0.0873526, -0.0982106, -0.1088938
    0.1637684, 0.1573717, 0.1507309, 0.1438743, 0.1368302, 0.1296271, 0.1222932, 0.1148570
    0.1073468, 0.0997909, 0.0922177, 0.0846556, 0.0771329, 0.0696779, 0.0623191, 0.0631225
    0.0604126, 0.0578293, 0.0553664, 0.0530178, 0.0507774, 0.0486393, 0.0465972, 0.0446453
    0.0427772, 0.0409871, 0.0392688, 0.0376163, 0.0360234, 0.0344842, 0.0758444, 0.0717167
    0.0675317, 0.0633012, 0.0590366, 0.0547495, 0.0504515, 0.0461541, 0.0418689, 0.0376074
    0.0333812, 0.0292018, 0.0250809, 0.0210299, 0.0170605, 0.0339686, 0.0336561, 0.0334516
    0.0333482, 0.0333392, 0.0334177, 0.0335770, 0.0338102, 0.0341105, 0.0344712, 0.0348853
    0.0353462, 0.0358469, 0.0363807, 0.0369408, 0.1753210, 0.1708903, 0.1662475, 0.1614031
    0.1563674, 0.1511509, 0.1457638, 0.1402166, 0.1345196, 0.1286833, 0.1227179, 0.1166339
    0.1104416, 0.1041514, 0.0977737, 0.1752777, 0.1731271, 0.1708030, 0.1683145, 0.1656706
    0.1628802, 0.1599522, 0.1568958, 0.1537198, 0.1504333, 0.1470452, 0.1435644, 0.1400000
    0.1363609, 0.1326562, 0.0577476, 0.0535079, 0.0492552, 0.0450018, 0.0407602, 0.0365426
    0.0323613, 0.0282287, 0.0241571, 0.0201588, 0.0162461, 0.0124313, 0.0087269, 0.0051450
    0.0016981, -0.0046913, -0.0047112, -0.0046630, -0.0045558, -0.0043984, -0.0041996, -0.0039682
    -0.0037132, -0.0034433, -0.0031675, -0.0028946, -0.0026334, -0.0023928, -0.0021816, -0.0020087
    0.0414634, 0.0404192, 0.0394774, 0.0386304, 0.0378704, 0.0371899, 0.0365810, 0.0360362
    0.0355478, 0.0351081, 0.0347094, 0.0343440, 0.0340044, 0.0336827, 0.0333714, 0.0304834
    0.0263261, 0.0222506, 0.0182734, 0.0144109, 0.0106797, 0.0070964, 0.0036773, 0.0004391
    -0.0026017, -0.0054286, -0.0080251, -0.0103746, -0.0124607, -0.0142668, 0.0169299, 0.0256628
    0.0345652, 0.0435966, 0.0527169, 0.0618855, 0.0710622, 0.0802066, 0.0892785, 0.0982373
    0.1070429, 0.1156548, 0.1240328, 0.1321364, 0.1399254, -0.0465299, -0.0475940, -0.0484199
    -0.0490128, -0.0493781, -0.0495209, -0.0494466, -0.0491604, -0.0486676, -0.0479734, -0.0470831
    -0.0460020, -0.0447354, -0.0432885, -0.0416666, 0.1927379, 0.1920820, 0.1912670, 0.1902912
    0.1891536, 0.1878529, 0.1863876, 0.1847566, 0.1829585, 0.1809921, 0.1788560, 0.1765489
    0.1740696, 0.1714167, 0.1685890, 0.0580951, 0.0636249, 0.0691058, 0.0745296, 0.0798881
    0.0851733, 0.0903771, 0.0954913, 0.1005077, 0.1054184, 0.1102151, 0.1148898, 0.1194344
    0.1238406, 0.1281005, 0.0756183, 0.0777809, 0.0802119, 0.0828844, 0.0857717, 0.0888471
    0.0920837, 0.0954548, 0.0989336, 0.1024933, 0.1061072, 0.1097486, 0.1133906, 0.1170065
    0.1205694, 0.1136137, 0.1113765, 0.1090580, 0.1066725, 0.1042345, 0.1017585, 0.0992589
    0.0967501, 0.0942468, 0.0917632, 0.0893139, 0.0869133, 0.0845760, 0.0823163, 0.0801487
    0.0915770, 0.0884047, 0.0851070, 0.0817012, 0.0782049, 0.0746354, 0.0710103, 0.0673470
    0.0636630, 0.0599756, 0.0563024, 0.0526608, 0.0490683, 0.0455423, 0.0421002, -0.0713279
    -0.0671417, -0.0627625, -0.0581976, -0.0534543, -0.0485400, -0.0434620, -0.0382276, -0.0328442
    -0.0273190, -0.0216595, -0.0158729, -0.0099667, -0.0039480, 0.0021757, 0.1376961, 0.1371807
    0.1364766, 0.1355716, 0.1344539, 0.1331114, 0.1315320, 0.1297038, 0.1276148, 0.1252529
    0.1226062, 0.1196625, 0.1164100, 0.1128366, 0.1089303, 0.0460724, 0.0474450, 0.0488383
    0.0502374, 0.0516272, 0.0529926, 0.0543187, 0.0555903, 0.0567924, 0.0579101, 0.0589281
    0.0598317, 0.0606056, 0.0612348, 0.0617044, 0.0942016, 0.0986613, 0.1031879, 0.1077696
    0.1123951, 0.1170525, 0.1217304, 0.1264171, 0.1311010, 0.1357706, 0.1404141, 0.1450200
    0.1495767, 0.1540726, 0.1584961, 0.0078228, 0.0080591, 0.0082836, 0.0085020, 0.0087199
    0.0089430, 0.0091768, 0.0094270, 0.0096993, 0.0099992, 0.0103325, 0.0107046, 0.0111214
    0.0115883, 0.0121110, 0.1244758, 0.1185586, 0.1126447, 0.1067364, 0.1008359, 0.0949453
    0.0890669, 0.0832028, 0.0773553, 0.0715264, 0.0657185, 0.0599336, 0.0541740, 0.0484419
    0.0427394, 0.0034125, 0.0052803, 0.0073446, 0.0095956, 0.0120235, 0.0146186, 0.0173711
    0.0202712, 0.0233091, 0.0264751, 0.0297593, 0.0331521, 0.0366435, 0.0402239, 0.0438835
    0.0285272, 0.0341139, 0.0396608, 0.0451516, 0.0505700, 0.0558996, 0.0611240, 0.0662269
    0.0711920, 0.0760029, 0.0806432, 0.0850966, 0.0893468, 0.0933774, 0.0971720, -0.0675938
    -0.0661418, -0.0645005, -0.0626812, -0.0606951, -0.0585537, -0.0562683, -0.0538501, -0.0513105
    -0.0486608, -0.0459123, -0.0430764, -0.0401643, -0.0371874, -0.0341571, 0.0736838, 0.0766777
    0.0797360, 0.0828606, 0.0860536, 0.0893170, 0.0926528, 0.0960631, 0.0995499, 0.1031153
    0.1067613, 0.1104900, 0.1143033, 0.1182034, 0.1221922, 0.1299862, 0.1206588, 0.1112411
    0.1017547, 0.0922212, 0.0826620, 0.0730988, 0.0635530, 0.0540461, 0.0445998, 0.0352355
    0.0259747, 0.0168390, 0.0078500, -0.0009709, -0.0291775, -0.0255162, -0.0217798, -0.0179731
    -0.0141011, -0.0101686, -0.0061806, -0.0021420, 0.0019424, 0.0060676, 0.0102287, 0.0144209
    0.0186391, 0.0228786, 0.0271344, -0.1157008, -0.1143829, -0.1130124, -0.1115773, -0.1100658
    -0.1084657, -0.1067652, -0.1049523, -0.1030151, -0.1009415, -0.0987197, -0.0963376, -0.0937833
    -0.0910449, -0.0881103, 0.0430258, 0.0483558, 0.0537198, 0.0591036, 0.0644927, 0.0698726
    0.0752292, 0.0805479, 0.0858144, 0.0910143, 0.0961332, 0.1011566, 0.1060703, 0.1108599
    0.1155109, 0.0235125, 0.0245434, 0.0255472, 0.0265204, 0.0274591, 0.0283597, 0.0292185
    0.0300317, 0.0307957, 0.0315067, 0.0321610, 0.0327550, 0.0332849, 0.0337469, 0.0341375
    -0.1055755, -0.1019250, -0.0981199, -0.0941612, -0.0900499, -0.0857871, -0.0813737, -0.0768110
    -0.0720999, -0.0672416, -0.0622369, -0.0570871, -0.0517931, -0.0463560, -0.0407769, 0.0199511
    0.0181087, 0.0161914, 0.0142142, 0.0121923, 0.0101409, 0.0080750, 0.0060098, 0.0039604
    0.0019421, -0.0000302, -0.0019412, -0.0037759, -0.0055191, -0.0071556, 0.0078183, 0.0163488
    0.0249356, 0.0335430, 0.0421357, 0.0506778, 0.0591339, 0.0674684, 0.0756457, 0.0836303
    0.0913864, 0.0988787, 0.1060714, 0.1129290, 0.1194159, 0.1175819, 0.1184317, 0.1192112
    0.1199168, 0.1205450, 0.1210922, 0.1215547, 0.1219290, 0.1222116, 0.1223987, 0.1224869
    0.1224725, 0.1223519, 0.1221216, 0.1217780, -0.0762521, -0.0726454, -0.0689160, -0.0650647
    -0.0610923, -0.0569998, -0.0527880, -0.0484579, -0.0440104, -0.0394463, -0.0347665, -0.0299720
    -0.0250636, -0.0200422, -0.0149087, 0.0802100, 0.0766074, 0.0728547, 0.0689609, 0.0649346
    0.0607848, 0.0565204, 0.0521502, 0.0476831, 0.0431280, 0.0384936, 0.0337889, 0.0290227
    0.0242040, 0.0193414, -0.0227196, -0.0175638, -0.0123160, -0.0069988, -0.0016349, 0.0037530
    0.0091424, 0.0145106, 0.0198349, 0.0250927, 0.0302613, 0.0353182, 0.0402406, 0.0450059
    0.0495916, 0.1171642, 0.1180332, 0.1189453, 0.1198711, 0.1207812, 0.1216461, 0.1224365
    0.1231229, 0.1236760, 0.1240663, 0.1242645, 0.1242410, 0.1239666, 0.1234118, 0.1225472
    0.1832776, 0.1791721, 0.1751167, 0.1711039, 0.1671267, 0.1631777, 0.1592499, 0.1553358
    0.1514284, 0.1475203, 0.1436044, 0.1396733, 0.1357200, 0.1317371, 0.1277175, 0.1764917
    0.1702412, 0.1638794, 0.1574249, 0.1508964, 0.1443125, 0.1376919, 0.1310533, 0.1244153
    0.1177966, 0.1112158, 0.1046916, 0.0982428, 0.0918878, 0.0856454, 0.0461447, 0.0472519
    0.0481896, 0.0489744, 0.0496233, 0.0501529, 0.0505800, 0.0509215, 0.0511942, 0.0514147
    0.0515999, 0.0517666, 0.0519315, 0.0521115, 0.0523233, 0.1171917, 0.1107748, 0.1041849
    0.0974353, 0.0905392, 0.0835099, 0.0763604, 0.0691039, 0.0617538, 0.0543231, 0.0468251
    0.0392730, 0.0316799, 0.0240590, 0.0164236, 0.1078465, 0.1062545, 0.1045919, 0.1028725
    0.1011103, 0.0993192, 0.0975132, 0.0957062, 0.0939122, 0.0921451, 0.0904188, 0.0887473
    0.0871446, 0.0856244, 0.0842009, 0.1429732, 0.1446297, 0.1460411, 0.1472248, 0.1481980
    0.1489781, 0.1495825, 0.1500285, 0.1503334, 0.1505147, 0.1505895, 0.1505753, 0.1504894
    0.1503491, 0.1501718, 0.0434268, 0.0348346, 0.0262183, 0.0176011, 0.0090055, 0.0004547
    -0.0080287, -0.0164216, -0.0247013, -0.0328449, -0.0408296, -0.0486323, -0.0562304, -0.0636009
    -0.0707209, 0.1558099, 0.1538810, 0.1518622, 0.1497529, 0.1475528, 0.1452614, 0.1428783
    0.1404030, 0.1378350, 0.1351740, 0.1324195, 0.1295710, 0.1266281, 0.1235904, 0.1204574
    0.0342500, 0.0376248, 0.0409424, 0.0442057, 0.0474180, 0.0505823, 0.0537017, 0.0567792
    0.0598179, 0.0628210, 0.0657914, 0.0687323, 0.0716468, 0.0745380, 0.0774088, 0.0213779
    0.0153543, 0.0092527, 0.0031022, -0.0030679, -0.0092285, -0.0153504, -0.0214043, -0.0273610
    -0.0331914, -0.0388662, -0.0443563, -0.0496324, -0.0546654, -0.0594259, 0.0250906, 0.0261104
    0.0270323, 0.0278646, 0.0286157, 0.0292938, 0.0299074, 0.0304647, 0.0309741, 0.0314441
    0.0318828, 0.0322987, 0.0327001, 0.0330953, 0.0334927, 0.0194744, 0.0216576, 0.0236223
    0.0253702, 0.0269032, 0.0282232, 0.0293320, 0.0302314, 0.0309233, 0.0314094, 0.0316918
    0.0317721, 0.0316523, 0.0313341, 0.0308195, 0.1507711, 0.1446761, 0.1384534, 0.1321168
    0.1256805, 0.1191586, 0.1125650, 0.1059140, 0.0992194, 0.0924955, 0.0857561, 0.0790155
    0.0722876, 0.0655866, 0.0589264, 0.0635858, 0.0671341, 0.0703689, 0.0732864, 0.0758829
    0.0781546, 0.0800977, 0.0817086, 0.0829834, 0.0839184, 0.0845099, 0.0847540, 0.0846472
    0.0841855, 0.0833653, 0.0628300, 0.0676506, 0.0724555, 0.0772423, 0.0820084, 0.0867513
    0.0914683, 0.0961570, 0.1008149, 0.1054393, 0.1100277, 0.1145777, 0.1190867, 0.1235520
    0.1279713, 0.0960708, 0.1061434, 0.1161268, 0.1260068, 0.1357697, 0.1454011, 0.1548872
    0.1642138, 0.1733670, 0.1823326, 0.1910966, 0.1996451, 0.2079639, 0.2160390, 0.2238564
    0.0014716, 0.0060123, 0.0106290, 0.0152982, 0.0199960, 0.0246986, 0.0293824, 0.0340236
    0.0385985, 0.0430833, 0.0474542, 0.0516877, 0.0557597, 0.0596467, 0.0633250, -0.0042423
    -0.0056001, -0.0069449, -0.0082871, -0.0096369, -0.0110047, -0.0124007, -0.0138353, -0.0153187
    -0.0168614, -0.0184734, -0.0201653, -0.0219472, -0.0238295, -0.0258224, 0.0333300, 0.0332461
    0.0331512, 0.0330440, 0.0329234, 0.0327884, 0.0326377, 0.0324702, 0.0322848, 0.0320804
    0.0318559, 0.0316100, 0.0313418, 0.0310499, 0.0307334, -0.0225802, -0.0192253, -0.0157104
    -0.0120457, -0.0082411, -0.0043066, -0.0002524, 0.0039115, 0.0081750, 0.0125282, 0.0169609
    0.0214632, 0.0260249, 0.0306360, 0.0352865, 0.0076610, 0.0087863, 0.0100086, 0.0113168
    0.0127000, 0.0141472, 0.0156472, 0.0171892, 0.0187621, 0.0203548, 0.0219564, 0.0235559
    0.0251422, 0.0267043, 0.0282313, -0.1738293, -0.1761017, -0.1782752, -0.1803391, -0.1822826
    -0.1840951, -0.1857657, -0.1872838, -0.1886386, -0.1898195, -0.1908155, -0.1916160, -0.1922104
    -0.1925877, -0.1927374, -0.0451716, -0.0459415, -0.0466503, -0.0473130, -0.0479450, -0.0485615
    -0.0491777, -0.0498087, -0.0504699, -0.0511765, -0.0519436, -0.0527865, -0.0537204, -0.0547606
    -0.0559223, 0.0313451, 0.0318530, 0.0323965, 0.0329620, 0.0335359, 0.0341042, 0.0346535
    0.0351699, 0.0356398, 0.0360494, 0.0363850, 0.0366330, 0.0367795, 0.0368111, 0.0367138
    -0.0629453, -0.0656955, -0.0683287, -0.0708379, -0.0732161, -0.0754561, -0.0775510, -0.0794936
    -0.0812770, -0.0828940, -0.0843376, -0.0856009, -0.0866766, -0.0875578, -0.0882374, 0.0367749
    0.0353453, 0.0339824, 0.0326986, 0.0315060, 0.0304169, 0.0294434, 0.0285978, 0.0278924
    0.0273393, 0.0269507, 0.0267389, 0.0267161, 0.0268945, 0.0272863, 0.0153616, 0.0136395
    0.0120974, 0.0107282, 0.0095248, 0.0084804, 0.0075878, 0.0068402, 0.0062305, 0.0057517
    0.0053969, 0.0051590, 0.0050310, 0.0050060, 0.0050769, -0.0192571, -0.0180364, -0.0167049
    -0.0152647, -0.0137180, -0.0120668, -0.0103133, -0.0084597, -0.0065079, -0.0044602, -0.0023187
    -0.0000854, 0.0022374, 0.0046478, 0.0071435, -0.0504750, -0.0500278, -0.0494339, -0.0486943
    -0.0478105, -0.0467836, -0.0456149, -0.0443057, -0.0428571, -0.0412705, -0.0395471, -0.0376881
    -0.0356948, -0.0335685, -0.0313103, 0.0913458, 0.0920834, 0.0927777, 0.0934243, 0.0940189
    0.0945571, 0.0950346, 0.0954470, 0.0957900, 0.0960592, 0.0962501, 0.0963585, 0.0963800
    0.0963102, 0.0961448, -0.0918816, -0.0955674, -0.0991570, -0.1026444, -0.1060237, -0.1092890
    -0.1124344, -0.1154539, -0.1183416, -0.1210915, -0.1236977, -0.1261543, -0.1284554, -0.1305949
    -0.1325670, -0.1254878, -0.1219582, -0.1183393, -0.1146367, -0.1108559, -0.1070026, -0.1030824
    -0.0991009, -0.0950638, -0.0909767, -0.0868450, -0.0826746, -0.0784710, -0.0742399, -0.0699867
    -0.0188197, -0.0160096, -0.0130668, -0.0099972, -0.0068067, -0.0035012, -0.0000866, 0.0034311
    0.0070461, 0.0107525, 0.0145442, 0.0184156, 0.0223605, 0.0263731, 0.0304476, -0.1910787
    -0.1908470, -0.1903828, -0.1896827, -0.1887434, -0.1875616, -0.1861340, -0.1844572, -0.1825280
    -0.1803431, -0.1778990, -0.1751926, -0.1722205, -0.1689794, -0.1654659, -0.0051557, -0.0135684
    -0.0221205, -0.0307969, -0.0395822, -0.0484611, -0.0574185, -0.0664390, -0.0755074, -0.0846083
    -0.0937265, -0.1028468, -0.1119539, -0.1210325, -0.1300673, 0.1134871, 0.1084404, 0.1031950
    0.0977655, 0.0921663, 0.0864123, 0.0805178, 0.0744976, 0.0683662, 0.0621382, 0.0558283
    0.0494509, 0.0430207, 0.0365523, 0.0300603, -0.1046408, -0.0965083, -0.0884417, -0.0804562
    -0.0725668, -0.0647887, -0.0571368, -0.0496262, -0.0422721, -0.0350896, -0.0280935, -0.0212992
    -0.0147215, -0.0083757, -0.0022768, -0.1469099, -0.1446536, -0.1423565, -0.1400080, -0.1375976
    -0.1351145, -0.1325483, -0.1298884, -0.1271242, -0.1242451, -0.1212405, -0.1180999, -0.1148126
    -0.1113682, -0.1077559, -0.1894790, -0.1789430, -0.1682553, -0.1574434, -0.1465348, -0.1355569
    -0.1245373, -0.1135035, -0.1024830, -0.0915034, -0.0805919, -0.0697763, -0.0590840, -0.0485425
    -0.0381794, 0.0206136, 0.0175415, 0.0142264, 0.0107152, 0.0070551, 0.0032930, -0.0005242
    -0.0043494, -0.0081356, -0.0118359, -0.0154033, -0.0187908, -0.0219514, -0.0248380, -0.0274038
    0.0076784, 0.0110569, 0.0141971, 0.0171045, 0.0197851, 0.0222446, 0.0244888, 0.0265233
    0.0283541, 0.0299868, 0.0314272, 0.0326811, 0.0337542, 0.0346523, 0.0353812, -0.1555190
    -0.1506316, -0.1457066, -0.1407458, -0.1357516, -0.1307259, -0.1256710, -0.1205889, -0.1154818
    -0.1103517, -0.1052009, -0.1000315, -0.0948455, -0.0896451, -0.0844324, -0.0116332, -0.0128253
    -0.0139098, -0.0148844, -0.0157466, -0.0164941, -0.0171244, -0.0176352, -0.0180240, -0.0182885
    -0.0184263, -0.0184349, -0.0183120, -0.0180551, -0.0176620, 0.0313084, 0.0215069, 0.0118641
    0.0024018, -0.0068584, -0.0158946, -0.0246852, -0.0332085, -0.0414426, -0.0493660, -0.0569567
    -0.0641932, -0.0710537, -0.0775165, -0.0835598, -0.2351192, -0.2378645, -0.2403578, -0.2425858
    -0.2445358, -0.2461946, -0.2475493, -0.2485869, -0.2492944, -0.2496587, -0.2496668, -0.2493059
    -0.2485628, -0.2474246, -0.2458783, -0.0743031, -0.0751638, -0.0758963, -0.0765045, -0.0769926
    -0.0773646, -0.0776245, -0.0777764, -0.0778244, -0.0777724, -0.0776245, -0.0773849, -0.0770575
    -0.0766464, -0.0761556, 0.0129456, 0.0108565, 0.0088393, 0.0068997, 0.0050435, 0.0032764
    0.0016040, 0.0000321, -0.0014336, -0.0027874, -0.0040236, -0.0051365, -0.0061204, -0.0069696
    -0.0076784, -0.0314597, -0.0340978, -0.0366073, -0.0389860, -0.0412320, -0.0433434, -0.0453180
    -0.0471540, -0.0488493, -0.0504018, -0.0518097, -0.0530709, -0.0541834, -0.0551452, -0.0559543
    -0.0195928, -0.0183120, -0.0171197, -0.0160205, -0.0150191, -0.0141201, -0.0133282, -0.0126480
    -0.0120842, -0.0116415, -0.0113244, -0.0111377, -0.0110861, -0.0111741, -0.0114064, -0.0014727
    -0.0040481, -0.0067013, -0.0094182, -0.0121844, -0.0149856, -0.0178075, -0.0206357, -0.0234560
    -0.0262541, -0.0290155, -0.0317262, -0.0343716, -0.0369375, -0.0394096, 0.0028188, 0.0025714
    0.0022344, 0.0018074, 0.0012896, 0.0006804, -0.0000208, -0.0008147, -0.0017019, -0.0026830
    -0.0037588, -0.0049297, -0.0061966, -0.0075599, -0.0090204, -0.1312037, -0.1342874, -0.1374081
    -0.1405464, -0.1436833, -0.1467993, -0.1498754, -0.1528924, -0.1558310, -0.1586720, -0.1613962
    -0.1639844, -0.1664174, -0.1686760, -0.1707409, -0.0834210, -0.0854099, -0.0872084, -0.0888062
    -0.0901933, -0.0913595, -0.0922946, -0.0929886, -0.0934314, -0.0936128, -0.0935226, -0.0931507
    -0.0924871, -0.0915216, -0.0902440, -0.1269360, -0.1238964, -0.1206035, -0.1170703, -0.1133097
    -0.1093350, -0.1051590, -0.1007948, -0.0962555, -0.0915540, -0.0867035, -0.0817170, -0.0766075
    -0.0713881, -0.0660717, -0.1243147, -0.1248381, -0.1253214, -0.1257477, -0.1260999, -0.1263611
    -0.1265145, -0.1265430, -0.1264298, -0.1261577, -0.1257100, -0.1250697, -0.1242198, -0.1231433
    -0.1218234, -0.1178561, -0.1159376, -0.1139148, -0.1117726, -0.1094960, -0.1070701, -0.1044797
    -0.1017098, -0.0987454, -0.0955715, -0.0921729, -0.0885346, -0.0846417, -0.0804791, -0.0760317
    0.1921535, 0.1888106, 0.1852842, 0.1815736, 0.1776784, 0.1735979, 0.1693315, 0.1648787
    0.1602388, 0.1554113, 0.1503955, 0.1451909, 0.1397969, 0.1342129, 0.1284383, -0.0805492
    -0.0816867, -0.0829022, -0.0841858, -0.0855277, -0.0869178, -0.0883464, -0.0898035, -0.0912792
    -0.0927637, -0.0942469, -0.0957191, -0.0971702, -0.0985905, -0.0999700, -0.0854903, -0.0839000
    -0.0822942, -0.0806689, -0.0790205, -0.0773450, -0.0756387, -0.0738976, -0.0721180, -0.0702960
    -0.0684278, -0.0665096, -0.0645375, -0.0625077, -0.0604164, -0.0130328, -0.0115379, -0.0101214
    -0.0087948, -0.0075694, -0.0064568, -0.0054684, -0.0046155, -0.0039097, -0.0033624, -0.0029850
    -0.0027890, -0.0027858, -0.0029867, -0.0034034, 0.0978079, 0.0932030, 0.0883645, 0.0833034
    0.0780305, 0.0725564, 0.0668922, 0.0610485, 0.0550361, 0.0488660, 0.0425489, 0.0360955
    0.0295168, 0.0228235, 0.0160264, -0.2308986, -0.2238554, -0.2166608, -0.2093216, -0.2018449
    -0.1942377, -0.1865069, -0.1786594, -0.1707023, -0.1626426, -0.1544871, -0.1462430, -0.1379171
    -0.1295165, -0.1210480, -0.0007219, 0.0001457, 0.0010045, 0.0018460, 0.0026619, 0.0034435
    0.0041826, 0.0048706, 0.0054992, 0.0060598, 0.0065441, 0.0069437, 0.0072500, 0.0074547
    0.0075492, 0.1608768, 0.1625552, 0.1639504, 0.1650570, 0.1658694, 0.1663821, 0.1665895
    0.1664860, 0.1660662, 0.1653244, 0.1642552, 0.1628531, 0.1611124, 0.1590276, 0.1565932
    -0.0862928, -0.0803660, -0.0744309, -0.0684965, -0.0625717, -0.0566656, -0.0507871, -0.0449452
    -0.0391491, -0.0334075, -0.0277296, -0.0221243, -0.0166006, -0.0111676, -0.0058342, -0.1001200
    -0.0950168, -0.0897929, -0.0844707, -0.0790729, -0.0736221, -0.0681406, -0.0626511, -0.0571762
    -0.0517384, -0.0463602, -0.0410641, -0.0358728, -0.0308088, -0.0258946, -0.1597874, -0.1543567
    -0.1486360, -0.1426434, -0.1363969, -0.1299145, -0.1232143, -0.1163143, -0.1092326, -0.1019871
    -0.0945960, -0.0870771, -0.0794487, -0.0717286, -0.0639350, 0.0122147, 0.0106612, 0.0088302
    0.0067486, 0.0044433, 0.0019410, -0.0007314, -0.0035470, -0.0064790, -0.0095006, -0.0125849
    -0.0157051, -0.0188344, -0.0219459, -0.0250128, -0.1619736, -0.1597414, -0.1576466, -0.1556759
    -0.1538160, -0.1520537, -0.1503755, -0.1487683, -0.1472186, -0.1457132, -0.1442387, -0.1427819
    -0.1413295, -0.1398681, -0.1383843, -0.2070564, -0.2003432, -0.1935624, -0.1867172, -0.1798110
    -0.1728471, -0.1658286, -0.1587589, -0.1516413, -0.1444790, -0.1372753, -0.1300334, -0.1227567
    -0.1154484, -0.1081117, -0.0875931, -0.0787133, -0.0696128, -0.0603182, -0.0508564, -0.0412539
    -0.0315375, -0.0217338, -0.0118696, -0.0019715, 0.0079337, 0.0178195, 0.0276589, 0.0374255
    0.0470925, 0.0289587, 0.0149135, 0.0008314, -0.0132465, -0.0272797, -0.0412271, -0.0550481
    -0.0687019, -0.0821475, -0.0953442, -0.1082512, -0.1208277, -0.1330329, -0.1448260, -0.1561660
    0.1237240, 0.1164677, 0.1092330, 0.1020420, 0.0949175, 0.0878817, 0.0809571, 0.0741661
    0.0675312, 0.0610748, 0.0548194, 0.0487873, 0.0430011, 0.0374831, 0.0322558, 0.1278310
    0.1184603, 0.1090755, 0.0996897, 0.0903158, 0.0809666, 0.0716550, 0.0623940, 0.0531964
    0.0440752, 0.0350433, 0.0261135, 0.0172988, 0.0086120, 0.0000662, 0.0870863, 0.0812047
    0.0752346, 0.0691859, 0.0630687, 0.0568931, 0.0506691, 0.0444067, 0.0381160, 0.0318071
    0.0254900, 0.0191747, 0.0128714, 0.0065899, 0.0003405, 0.1446231, 0.1462580, 0.1478367
    0.1493495, 0.1507866, 0.1521383, 0.1533950, 0.1545469, 0.1555842, 0.1564974, 0.1572765
    0.1579120, 0.1583940, 0.1587130, 0.1588590, 0.2532810, 0.2510079, 0.2485122, 0.2457846
    0.2428154, 0.2395953, 0.2361147, 0.2323641, 0.2283340, 0.2240149, 0.2193973, 0.2144718
    0.2092287, 0.2036587, 0.1977522, 0.1064963, 0.1043648, 0.1021136, 0.0997456, 0.0972637
    0.0946709, 0.0919698, 0.0891635, 0.0862548, 0.0832465, 0.0801415, 0.0769428, 0.0736531
    0.0702754, 0.0668124, 0.0679999, 0.0705212, 0.0731146, 0.0757513, 0.0784027, 0.0810399
    0.0836342, 0.0861569, 0.0885794, 0.0908727, 0.0930083, 0.0949574, 0.0966912, 0.0981810
    0.0993982, 0.1628666, 0.1595736, 0.1559618, 0.1520444, 0.1478353, 0.1433479, 0.1385958
    0.1335926, 0.1283518, 0.1228871, 0.1172118, 0.1113397, 0.1052843, 0.0990592, 0.0926779
    0.1077648, 0.1016812, 0.0954430, 0.0890764, 0.0826073, 0.0760617, 0.0694655, 0.0628449
    0.0562257, 0.0496339, 0.0430956, 0.0366366, 0.0302831, 0.0240609, 0.0179962, -0.0468305
    -0.0464947, -0.0460247, -0.0454217, -0.0446865, -0.0438203, -0.0428241, -0.0416990, -0.0404459
    -0.0390659, -0.0375601, -0.0359295, -0.0341752, -0.0322981, -0.0302994, -0.0855380, -0.0826550
    -0.0795974, -0.0763788, -0.0730125, -0.0695120, -0.0658909, -0.0621624, -0.0583401, -0.0544374
    -0.0504678, -0.0464448, -0.0423817, -0.0382921, -0.0341893, -0.0045786, 0.0024305, 0.0097509
    0.0173568, 0.0252219, 0.0333204, 0.0416262, 0.0501132, 0.0587555, 0.0675270, 0.0764016
    0.0853535, 0.0943565, 0.1033846, 0.1124118, 0.0050013, 0.0087047, 0.0123087, 0.0158091
    0.0192014, 0.0224811, 0.0256438, 0.0286851, 0.0316005, 0.0343856, 0.0370361, 0.0395474
    0.0419151, 0.0441348, 0.0462021, -0.1196664, -0.1153921, -0.1110270, -0.1065804, -0.1020619
    -0.0974809, -0.0928469, -0.0881694, -0.0834578, -0.0787215, -0.0739701, -0.0692130, -0.0644596
    -0.0597195, -0.0550021, 0.1051292, 0.1014501, 0.0977800, 0.0941162, 0.0904563, 0.0867979
    0.0831385, 0.0794756, 0.0758067, 0.0721294, 0.0684412, 0.0647397, 0.0610223, 0.0572866
    0.0535301, -0.0808895, -0.0778422, -0.0747161, -0.0715174, -0.0682524, -0.0649272, -0.0615482
    -0.0581216, -0.0546536, -0.0511504, -0.0476184, -0.0440637, -0.0404927, -0.0369114, -0.0333263
    0.0999047, 0.0989664, 0.0977657, 0.0963056, 0.0945895, 0.0926205, 0.0904017, 0.0879363
    0.0852275, 0.0822784, 0.0790923, 0.0756722, 0.0720214, 0.0681430, 0.0640402, -0.0022803
    0.0026598, 0.0078019, 0.0131314, 0.0186336, 0.0242941, 0.0300981, 0.0360311, 0.0420785
    0.0482256, 0.0544579, 0.0607607, 0.0671194, 0.0735195, 0.0799463, 0.0829340, 0.0891417
    0.0952623, 0.1012705, 0.1071413, 0.1128497, 0.1183705, 0.1236787, 0.1287493, 0.1335570
    0.1380769, 0.1422840, 0.1461530, 0.1496591, 0.1527769, -0.0295851, -0.0252719, -0.0208426
    -0.0163025, -0.0116570, -0.0069118, -0.0020721, 0.0028565, 0.0078685, 0.0129585, 0.0181210
    0.0233507, 0.0286419, 0.0339893, 0.0393874, 0.0483219, 0.0474391, 0.0466362, 0.0459146
    0.0452755, 0.0447203, 0.0442503, 0.0438669, 0.0435714, 0.0433652, 0.0432496, 0.0432258
    0.0432954, 0.0434595, 0.0437196, 0.0822043, 0.0850044, 0.0876840, 0.0902413, 0.0926743
    0.0949810, 0.0971595, 0.0992080, 0.1011243, 0.1029067, 0.1045532, 0.1060618, 0.1074307
    0.1086577, 0.1097412, 0.0338109, 0.0335702, 0.0332464, 0.0328478, 0.0323830, 0.0318602
    0.0312877, 0.0306741, 0.0300275, 0.0293566, 0.0286694, 0.0279746, 0.0272804, 0.0265951
    0.0259273, 0.0483928, 0.0520914, 0.0555820, 0.0588686, 0.0619551, 0.0648455, 0.0675438
    0.0700539, 0.0723798, 0.0745255, 0.0764948, 0.0782919, 0.0799206, 0.0813848, 0.0826886
    -0.0806028, -0.0702249, -0.0598241, -0.0494176, -0.0390226, -0.0286561, -0.0183354, -0.0080776
    0.0021001, 0.0121805, 0.0221466, 0.0319811, 0.0416668, 0.0511867, 0.0605236, -0.1056136
    -0.1041221, -0.1025624, -0.1009245, -0.0991982, -0.0973734, -0.0954399, -0.0933877, -0.0912066
    -0.0888864, -0.0864170, -0.0837883, -0.0809902, -0.0780125, -0.0748451, -0.0049842, -0.0036401
    -0.0022441, -0.0007943, 0.0007110, 0.0022738, 0.0038959, 0.0055792, 0.0073256, 0.0091369
    0.0110150, 0.0129617, 0.0149790, 0.0170687, 0.0192327, 0.1909152, 0.1798323, 0.1686236
    0.1573088, 0.1459077, 0.1344398, 0.1229250, 0.1113830, 0.0998334, 0.0882960, 0.0767904
    0.0653364, 0.0539538, 0.0426621, 0.0314812, 0.0252666, 0.0249688, 0.0246618, 0.0243544
    0.0240557, 0.0237746, 0.0235200, 0.0233009, 0.0231263, 0.0230051, 0.0229463, 0.0229588
    0.0230515, 0.0232335, 0.0235137, 0.0518931, 0.0576313, 0.0633168, 0.0689476, 0.0745214
    0.0800360, 0.0854892, 0.0908789, 0.0962028, 0.1014588, 0.1066445, 0.1117580, 0.1167969
    0.1217591, 0.1266424, 0.2258873, 0.2296284, 0.2332051, 0.2366264, 0.2399011, 0.2430383
    0.2460469, 0.2489358, 0.2517139, 0.2543902, 0.2569735, 0.2594729, 0.2618972, 0.2642555
    0.2665566, 0.2044941, 0.2021081, 0.1997304, 0.1973543, 0.1949737, 0.1925821, 0.1901732
    0.1877406, 0.1852779, 0.1827787, 0.1802367, 0.1776455, 0.1749987, 0.1722899, 0.1695128
    0.0560720, 0.0525972, 0.0492163, 0.0459392, 0.0427757, 0.0397355, 0.0368284, 0.0340642
    0.0314527, 0.0290036, 0.0267268, 0.0246319, 0.0227289, 0.0210274, 0.0195373, 0.1913830
    0.1890865, 0.1866932, 0.1842067, 0.1816307, 0.1789685, 0.1762239, 0.1734003, 0.1705012
    0.1675303, 0.1644911, 0.1613871, 0.1582219, 0.1549989, 0.1517219, 0.1230551, 0.1219464
    0.1208935, 0.1199050, 0.1189900, 0.1181571, 0.1174153, 0.1167733, 0.1162400, 0.1158242
    0.1155346, 0.1153802, 0.1153698, 0.1155122, 0.1158162, 0.2690834, 0.2658933, 0.2625576
    0.2590834, 0.2554776, 0.2517473, 0.2478996, 0.2439415, 0.2398800, 0.2357221, 0.2314748
    0.2271453, 0.2227404, 0.2182674, 0.2137331, 0.2457059, 0.2494594, 0.2529362, 0.2561381
    0.2590666, 0.2617236, 0.2641108, 0.2662298, 0.2680824, 0.2696702, 0.2709950, 0.2720585
    0.2728624, 0.2734084, 0.2736982, 0.0889433, 0.0895808, 0.0901462, 0.0906389, 0.0910583
    0.0914039, 0.0916752, 0.0918715, 0.0919923, 0.0920371, 0.0920053, 0.0918964, 0.0917097
    0.0914448, 0.0911010, 0.1214404, 0.1181914, 0.1149008, 0.1115753, 0.1082218, 0.1048470
    0.1014577, 0.0980608, 0.0946629, 0.0912709, 0.0878915, 0.0845316, 0.0811979, 0.0778972
    0.0746362, 0.1312768, 0.1341929, 0.1370061, 0.1397157, 0.1423206, 0.1448200, 0.1472131
    0.1494988, 0.1516763, 0.1537446, 0.1557029, 0.1575503, 0.1592859, 0.1609087, 0.1624179
    -0.1911697, -0.1828597, -0.1743380, -0.1656268, -0.1567489, -0.1477265, -0.1385823, -0.1293386
    -0.1200181, -0.1106431, -0.1012362, -0.0918198, -0.0824165, -0.0730487, -0.0637388, 0.2315037
    0.2286144, 0.2255547, 0.2223347, 0.2189648, 0.2154552, 0.2118163, 0.2080584, 0.2041916
    0.2002264, 0.1961730, 0.1920416, 0.1878426, 0.1835863, 0.1792830, 0.0178467, 0.0132863
    0.0087795, 0.0043292, -0.0000618, -0.0043908, -0.0086548, -0.0128510, -0.0169767, -0.0210290
    -0.0250051, -0.0289022, -0.0327175, -0.0364481, -0.0400912, -0.0051967, 0.0002137, 0.0056483
    0.0111066, 0.0165880, 0.0220920, 0.0276180, 0.0331656, 0.0387341, 0.0443230, 0.0499318
    0.0555599, 0.0612068, 0.0668720, 0.0725548, -0.0534128, -0.0469931, -0.0403231, -0.0334253
    -0.0263222, -0.0190363, -0.0115900, -0.0040059, 0.0036937, 0.0114863, 0.0193493, 0.0272603
    0.0351968, 0.0431365, 0.0510566, 0.1588127, 0.1562264, 0.1535381, 0.1507502, 0.1478653
    0.1448859, 0.1418147, 0.1386540, 0.1354065, 0.1320747, 0.1286612, 0.1251684, 0.1215990
    0.1179555, 0.1142404, -0.0196346, -0.0122905, -0.0048771, 0.0025812, 0.0100603, 0.0175356
    0.0249829, 0.0323779, 0.0396961, 0.0469133, 0.0540052, 0.0609473, 0.0677154, 0.0742851
    0.0806320, -0.0194547, -0.0144593, -0.0093448, -0.0041272, 0.0011776, 0.0065535, 0.0119844
    0.0174545, 0.0229476, 0.0284478, 0.0339390, 0.0394053, 0.0448307, 0.0501990, 0.0554944
    0.2149450, 0.2089208, 0.2028573, 0.1967555, 0.1906165, 0.1844415, 0.1782315, 0.1719877
    0.1657113, 0.1594033, 0.1530648, 0.1466970, 0.1403010, 0.1338779, 0.1274289, 0.2727118
    0.2707212, 0.2684312, 0.2658577, 0.2630167, 0.2599243, 0.2565964, 0.2530489, 0.2492979
    0.2453593, 0.2412491, 0.2369832, 0.2325778, 0.2280487, 0.2234119, 0.2908449, 0.2864383
    0.2819546, 0.2773974, 0.2727706, 0.2680777, 0.2633227, 0.2585091, 0.2536408, 0.2487215
    0.2437548, 0.2387446, 0.2336945, 0.2286083, 0.2234898, 0.1203519, 0.1176529, 0.1150360
    0.1124964, 0.1100295, 0.1076304, 0.1052944, 0.1030168, 0.1007928, 0.0986177, 0.0964867
    0.0943950, 0.0923380, 0.0903108, 0.0883088, 0.1342596, 0.1296648, 0.1250142, 0.1203250
    0.1156146, 0.1109004, 0.1061997, 0.1015299, 0.0969084, 0.0923524, 0.0878795, 0.0835068
    0.0792518, 0.0751319, 0.0711643, 0.0955426, 0.0947638, 0.0940026, 0.0932464, 0.0924826
    0.0916986, 0.0908817, 0.0900194, 0.0890989, 0.0881078, 0.0870332, 0.0858628, 0.0845838
    0.0831836, 0.0816496, 0.2465685, 0.2458470, 0.2449062, 0.2437551, 0.2424026, 0.2408576
    0.2391289, 0.2372257, 0.2351567, 0.2329309, 0.2305571, 0.2280444, 0.2254016, 0.2226378
    0.2197616, 0.0794464, 0.0864959, 0.0934336, 0.1002606, 0.1069784, 0.1135880, 0.1200909
    0.1264883, 0.1327813, 0.1389714, 0.1450596, 0.1510475, 0.1569361, 0.1627267, 0.1684207
    0.1963171, 0.1886084, 0.1809510, 0.1733500, 0.1658103, 0.1583369, 0.1509345, 0.1436082
    0.1363630, 0.1292036, 0.1221351, 0.1151623, 0.1082902, 0.1015238, 0.0948679, 0.2474076
    0.2408282, 0.2341390, 0.2273431, 0.2204438, 0.2134445, 0.2063484, 0.1991587, 0.1918788
    0.1845119, 0.1770613, 0.1695302, 0.1619219, 0.1542397, 0.1464869, 0.2076822, 0.2012793
    0.1948858, 0.1884997, 0.1821190, 0.1757418, 0.1693661, 0.1629898, 0.1566111, 0.1502278
    0.1438380, 0.1374397, 0.1310309, 0.1246097, 0.1181739, 0.0658510, 0.0682835, 0.0707382
    0.0732091, 0.0756898, 0.0781742, 0.0806561, 0.0831292, 0.0855873, 0.0880241, 0.0904336
    0.0928094, 0.0951454, 0.0974352, 0.0996728, 0.1487795, 0.1482999, 0.1477089, 0.1470036
    0.1461812, 0.1452389, 0.1441739, 0.1429835, 0.1416647, 0.1402150, 0.1386314, 0.1369111
    0.1350514, 0.1330495, 0.1309025, 0.1061712, 0.1075576, 0.1089078, 0.1102219, 0.1115002
    0.1127430, 0.1139504, 0.1151226, 0.1162600, 0.1173626, 0.1184307, 0.1194646, 0.1204645
    0.1214305, 0.1223629, 0.1454733, 0.1463719, 0.1472723, 0.1481596, 0.1490188, 0.1498352
    0.1505940, 0.1512802, 0.1518790, 0.1523757, 0.1527552, 0.1530028, 0.1531036, 0.1530429
    0.1528056, -0.0231427, -0.0202108, -0.0171239, -0.0138840, -0.0104929, -0.0069524, -0.0032644
    0.0005694, 0.0045470, 0.0086665, 0.0129263, 0.0173243, 0.0218589, 0.0265280, 0.0313299
    0.2332528, 0.2245113, 0.2156977, 0.2068252, 0.1979070, 0.1889566, 0.1799872, 0.1710121
    0.1620444, 0.1530976, 0.1441849, 0.1353196, 0.1265149, 0.1177841, 0.1091406, 0.1224493
    0.1205608, 0.1187535, 0.1170306, 0.1153955, 0.1138515, 0.1124017, 0.1110496, 0.1097983
    0.1086513, 0.1076116, 0.1066827, 0.1058678, 0.1051702, 0.1045932, 0.1664257, 0.1639612
    0.1615259, 0.1591250, 0.1567638, 0.1544478, 0.1521824, 0.1499728, 0.1478244, 0.1457426
    0.1437328, 0.1418003, 0.1399504, 0.1381886, 0.1365202, -0.0645844, -0.0611641, -0.0576941
    -0.0541865, -0.0506532, -0.0471064, -0.0435581, -0.0400202, -0.0365049, -0.0330241, -0.0295900
    -0.0262145, -0.0229096, -0.0196874, -0.0165600, 0.2161816, 0.2150876, 0.2137645, 0.2122285
    0.2104957, 0.2085822, 0.2065042, 0.2042779, 0.2019194, 0.1994449, 0.1968704, 0.1942121
    0.1914863, 0.1887090, 0.1858965, 0.0459910, 0.0515672, 0.0571843, 0.0628183, 0.0684450
    0.0740403, 0.0795800, 0.0850400, 0.0903962, 0.0956245, 0.1007006, 0.1056005, 0.1103000
    0.1147751, 0.1190015, 0.0834918, 0.0814506, 0.0793134, 0.0770865, 0.0747765, 0.0723897
    0.0699327, 0.0674119, 0.0648337, 0.0622046, 0.0595310, 0.0568194, 0.0540763, 0.0513081
    0.0485212, 0.0777290, 0.0844190, 0.0911303, 0.0978574, 0.1045951, 0.1113379, 0.1180807
    0.1248179, 0.1315444, 0.1382547, 0.1449436, 0.1516057, 0.1582357, 0.1648283, 0.1713781
    0.1196171, 0.1229443, 0.1260704, 0.1289904, 0.1316994, 0.1341928, 0.1364655, 0.1385127
    0.1403294, 0.1419110, 0.1432523, 0.1443487, 0.1451952, 0.1457870, 0.1461191, -0.0283099
    -0.0327551, -0.0369110, -0.0407789, -0.0443603, -0.0476565, -0.0506688, -0.0533986, -0.0558472
    -0.0580159, -0.0599061, -0.0615192, -0.0628565, -0.0639194, -0.0647091, 0.1341761, 0.1328827
    0.1314290, 0.1298132, 0.1280332, 0.1260872, 0.1239730, 0.1216889, 0.1192328, 0.1166027
    0.1137967, 0.1108128, 0.1076492, 0.1043037, 0.1007745, 0.1416419, 0.1427703, 0.1437053
    0.1444388, 0.1449628, 0.1452693, 0.1453504, 0.1451981, 0.1448042, 0.1441609, 0.1432602
    0.1420940, 0.1406543, 0.1389332, 0.1369226, 0.1869225, 0.1868909, 0.1866248, 0.1861433
    0.1854657, 0.1846113, 0.1835993, 0.1824490, 0.1811796, 0.1798103, 0.1783604, 0.1768492
    0.1752959, 0.1737198, 0.1721401, -0.0069202, -0.0002762, 0.0062697, 0.0127071, 0.0190255
    0.0252145, 0.0312638, 0.0371628, 0.0429012, 0.0484685, 0.0538543, 0.0590482, 0.0640397
    0.0688185, 0.0733741, -0.1575498, -0.1507276, -0.1437414, -0.1366053, -0.1293336, -0.1219406
    -0.1144405, -0.1068475, -0.0991758, -0.0914397, -0.0836534, -0.0758312, -0.0679872, -0.0601358
    -0.0522911, -0.0665018, -0.0665651, -0.0666498, -0.0667266, -0.0667661, -0.0667391, -0.0666161
    -0.0663678, -0.0659649, -0.0653781, -0.0645780, -0.0635353, -0.0622206, -0.0606047, -0.0586581
    0.0706061, 0.0781613, 0.0856021, 0.0929083, 0.1000596, 0.1070357, 0.1138165, 0.1203818
    0.1267111, 0.1327844, 0.1385814, 0.1440819, 0.1492655, 0.1541121, 0.1586015, -0.0548076
    -0.0547272, -0.0545126, -0.0541620, -0.0536739, -0.0530464, -0.0522780, -0.0513669, -0.0503114
    -0.0491099, -0.0477607, -0.0462620, -0.0446122, -0.0428095, -0.0408524, -0.0829585, -0.0872601
    -0.0915451, -0.0957955, -0.0999938, -0.1041221, -0.1081627, -0.1120980, -0.1159102, -0.1195815
    -0.1230942, -0.1264306, -0.1295730, -0.1325036, -0.1352047, 0.1853649, 0.1759496, 0.1665995
    0.1573244, 0.1481340, 0.1390382, 0.1300467, 0.1211692, 0.1124154, 0.1037952, 0.0953183
    0.0869944, 0.0788333, 0.0708448, 0.0630386, 0.1070912, 0.1070212, 0.1069912, 0.1069867
    0.1069930, 0.1069958, 0.1069804, 0.1069322, 0.1068367, 0.1066794, 0.1064456, 0.1061210
    0.1056908, 0.1051406, 0.1044558, 0.2722675, 0.2657644, 0.2590891, 0.2522559, 0.2452796
    0.2381749, 0.2309564, 0.2236387, 0.2162364, 0.2087644, 0.2012370, 0.1936691, 0.1860752
    0.1784700, 0.1708681, 0.0379722, 0.0371302, 0.0364627, 0.0359465, 0.0355583, 0.0352749
    0.0350730, 0.0349293, 0.0348207, 0.0347238, 0.0346154, 0.0344723, 0.0342711, 0.0339887
    0.0336017, 0.2129385, 0.2123367, 0.2116180, 0.2107780, 0.2098128, 0.2087179, 0.2074893
    0.2061225, 0.2046136, 0.2029582, 0.2011520, 0.1991909, 0.1970707, 0.1947872, 0.1923360
    0.1535310, 0.1482175, 0.1427947, 0.1372636, 0.1316254, 0.1258812, 0.1200321, 0.1140793
    0.1080238, 0.1018669, 0.0956095, 0.0892529, 0.0827982, 0.0762464, 0.0695987, 0.0699391
    0.0717561, 0.0734965, 0.0751559, 0.0767302, 0.0782152, 0.0796065, 0.0808998, 0.0820911
    0.0831760, 0.0841502, 0.0850095, 0.0857497, 0.0863665, 0.0868557, 0.0558981, 0.0520828
    0.0482006, 0.0442614, 0.0402750, 0.0362514, 0.0322005, 0.0281320, 0.0240558, 0.0199819
    0.0159201, 0.0118802, 0.0078722, 0.0039058, -0.0000090, 0.0808436, 0.0811768, 0.0814743
    0.0817324, 0.0819469, 0.0821141, 0.0822299, 0.0822905, 0.0822918, 0.0822300, 0.0821011
    0.0819012, 0.0816264, 0.0812726, 0.0808361, 0.0998646, 0.1001313, 0.1004008, 0.1006599
    0.1008952, 0.1010937, 0.1012419, 0.1013266, 0.1013347, 0.1012528, 0.1010677, 0.1007661
    0.1003349, 0.0997606, 0.0990302, 0.1060394, 0.1010311, 0.0958384, 0.0904839, 0.0849906
    0.0793812, 0.0736786, 0.0679056, 0.0620850, 0.0562397, 0.0503924, 0.0445661, 0.0387835
    0.0330674, 0.0274408, 0.2332947, 0.2320427, 0.2308875, 0.2298162, 0.2288162, 0.2278747
    0.2269789, 0.2261161, 0.2252734, 0.2244383, 0.2235978, 0.2227393, 0.2218500, 0.2209171
    0.2199278, 0.0550572, 0.0569540, 0.0587321, 0.0604078, 0.0619976, 0.0635183, 0.0649862
    0.0664179, 0.0678300, 0.0692390, 0.0706614, 0.0721138, 0.0736127, 0.0751746, 0.0768160
    -0.0149594, -0.0108012, -0.0064672, -0.0019757, 0.0026552, 0.0074075, 0.0122629, 0.0172033
    0.0222107, 0.0272668, 0.0323535, 0.0374528, 0.0425464, 0.0476162, 0.0526442, 0.1750945
    0.1769665, 0.1787075, 0.1803229, 0.1818182, 0.1831989, 0.1844704, 0.1856382, 0.1867078
    0.1876846, 0.1885740, 0.1893816, 0.1901128, 0.1907730, 0.1913678, 0.1975685, 0.1951428
    0.1925752, 0.1898648, 0.1870113, 0.1840140, 0.1808723, 0.1775856, 0.1741533, 0.1705749
    0.1668496, 0.1629769, 0.1589562, 0.1547870, 0.1504685, -0.0795670, -0.0729030, -0.0660391
    -0.0589958, -0.0517936, -0.0444528, -0.0369940, -0.0294375, -0.0218038, -0.0141132, -0.0063864
    0.0013565, 0.0090948, 0.0168082, 0.0244762, 0.0386637, 0.0421957, 0.0456294, 0.0489788
    0.0522580, 0.0554809, 0.0586617, 0.0618143, 0.0649528, 0.0680911, 0.0712434, 0.0744237
    0.0776459, 0.0809242, 0.0842725, 0.1762898, 0.1734540, 0.1707227, 0.1680910, 0.1655543
    0.1631078, 0.1607467, 0.1584662, 0.1562618, 0.1541284, 0.1520615, 0.1500562, 0.1481079
    0.1462117, 0.1443628, 0.1414204, 0.1420275, 0.1424706, 0.1427564, 0.1428914, 0.1428824
    0.1427360, 0.1424588, 0.1420574, 0.1415386, 0.1409089, 0.1401750, 0.1393435, 0.1384210
    0.1374143, 0.0507742, 0.0516949, 0.0525954, 0.0534699, 0.0543126, 0.0551177, 0.0558795
    0.0565920, 0.0572496, 0.0578463, 0.0583765, 0.0588343, 0.0592140, 0.0595096, 0.0597156
    0.1212202, 0.1248918, 0.1285754, 0.1322461, 0.1358794, 0.1394503, 0.1429341, 0.1463062
    0.1495416, 0.1526156, 0.1555035, 0.1581806, 0.1606220, 0.1628030, 0.1646989, 0.0767328
    0.0764263, 0.0761055, 0.0757784, 0.0754530, 0.0751374, 0.0748396, 0.0745677, 0.0743298
    0.0741338, 0.0739877, 0.0738998, 0.0738779, 0.0739301, 0.0740645, -0.0536897, -0.0532007
    -0.0526201, -0.0519434, -0.0511661, -0.0502836, -0.0492915, -0.0481853, -0.0469603, -0.0456121
    -0.0441361, -0.0425279, -0.0407828, -0.0388965, -0.0368642, 0.0710855, 0.0700342, 0.0690583
    0.0681560, 0.0673251, 0.0665637, 0.0658696, 0.0652410, 0.0646758, 0.0641719, 0.0637273
    0.0633401, 0.0630081, 0.0627294, 0.0625020, 0.0808554, 0.0854375, 0.0900328, 0.0946292
    0.0992150, 0.1037781, 0.1083068, 0.1127890, 0.1172130, 0.1215668, 0.1258384, 0.1300161
    0.1340879, 0.1380419, 0.1418661, 0.0693192, 0.0700511, 0.0708074, 0.0715877, 0.0723916
    0.0732187, 0.0740684, 0.0749404, 0.0758342, 0.0767494, 0.0776856, 0.0786423, 0.0796191
    0.0806156, 0.0816313, -0.0169127, -0.0209404, -0.0248180, -0.0285401, -0.0321018, -0.0354976
    -0.0387223, -0.0417708, -0.0446378, -0.0473180, -0.0498062, -0.0520972, -0.0541858, -0.0560667
    -0.0577347, 0.1443522, 0.1401007, 0.1358542, 0.1316094, 0.1273627, 0.1231108, 0.1188502
    0.1145773, 0.1102889, 0.1059814, 0.1016513, 0.0972953, 0.0929098, 0.0884914, 0.0840367];

   // MatMul 'l0_base': W(16×28) + b(16)
   w2 : ARRAY[0..463] OF REAL :=
[0.3825108, 0.0485370, 0.1553129, -0.0322751, -0.0784649, -0.0979913, 0.0300957, 0.0884262
    0.4441010, 0.4753721, 0.0841905, 0.5709860, -0.1169512, 0.0279510, -0.4520210, 0.0597628
    -0.0623482, 0.3703407, 0.2142555, -0.0983415, 0.1050850, -0.1663091, 0.0088212, 0.4195257
    0.1522815, 0.1986880, 0.1510919, -0.1282427, 0.3712382, 0.1146060, 0.1542422, 0.1171126
    0.2055789, 0.3519945, 0.0072344, -0.0827091, 0.3385513, -0.0698119, -0.2152457, -0.2510968
    -0.0464614, 0.2837242, 0.1521953, -0.2826805, 0.2372488, 0.2268303, -0.0034563, -0.3720433
    0.2629979, 0.2415776, 0.3191497, -0.2184810, 0.3111473, -0.0105020, 0.0376962, 0.1190158
    0.3232971, 0.4169890, 0.5698181, -0.1865906, -0.3292018, -0.0329375, 0.2244749, 0.0721402
    -0.0152652, -0.0166362, 0.3252053, 0.6891209, -0.0415161, 0.1034102, -0.3547171, -0.2161654
    -0.4391139, 0.4122617, 0.0130419, 0.1791824, 0.1126268, -0.2466755, -0.1145965, 0.4281023
    -0.0451292, -0.0343471, 0.2910257, -0.2015965, 0.0736524, -0.1599241, -0.1555228, 0.1631235
    0.4105036, 0.0649687, 0.0696781, -0.0144990, 0.0322124, -0.2427009, 0.0216245, -0.3794920
    0.2226683, 0.0153569, 0.5966946, 0.2662281, 0.1313384, -0.2857246, 0.1990728, 0.2923056
    -0.1706078, 0.0431573, -0.0784950, -0.4066874, 0.2723872, -0.0669259, -0.1014354, 0.1851601
    0.1155580, 0.0328991, -0.1228462, 0.3848465, 0.1363740, 0.2065286, -0.2832288, 0.1447309
    0.3049465, 0.3290030, -0.2855318, -0.0919528, -0.3483118, 0.2557819, 0.0905260, -0.2083652
    -0.0865834, 0.1593322, -0.3704533, -0.3512432, 0.1130393, -0.0451635, 0.2307400, 0.2154467
    -0.2300902, 0.2571728, 0.0086791, -0.0826596, 0.2138963, -0.0882278, -0.3927259, 0.4067457
    0.5467825, 0.0519261, -0.1621639, 0.0754226, 0.3409606, -0.4424310, -0.1752899, -0.6468470
    -0.4518577, 0.1852804, 0.5239546, -0.4837608, 0.2453886, 0.0739599, 0.2208461, -0.0689023
    0.1996087, 0.2635212, 0.2272361, -0.2062375, 0.0911828, -0.2152853, 0.0327323, 0.4654786
    0.2093491, 0.3581172, 0.2059541, -0.3333091, 0.2941960, -0.3455873, 0.4597460, -0.1189834
    0.0614193, -0.2540230, -0.0933914, -0.1069163, -0.0233051, 0.0415943, -0.1575655, -0.1822143
    -0.0055236, 0.1665109, 0.2270915, 0.1261556, -0.1864877, 0.1021470, -0.5130386, -0.0406230
    0.2724753, -0.1806795, -0.2065981, 0.3496896, -0.0389578, 0.1853916, 0.2067362, -0.1305270
    -0.3989385, -0.1613440, 0.2444519, -0.0867275, -0.0449195, 0.3072193, 0.2403889, 0.7019656
    0.4396943, -0.0941337, -0.5315250, 0.5334889, -0.1114494, 0.0906655, -0.0945825, 0.0411999
    -0.3302798, 0.0001274, -0.2760554, 0.4839795, -0.1854450, 0.4298583, 0.1623260, -0.3952270
    0.1250749, 0.1666509, 0.1406655, -0.1982276, -0.6801189, -0.2674226, -0.1567214, 0.0115039
    0.2678978, 0.3268091, -0.0339156, 0.3136737, -0.2586173, -0.0368428, -0.3921259, -0.2594979
    -0.1625591, 0.2014341, -0.3031742, -0.4860181, 0.3265654, 0.1123224, -0.0007127, 0.4288552
    -0.0741221, 0.0886679, 0.1864470, -0.0907285, 0.3239636, 0.1910028, 0.0061336, 0.1117132
    0.2615147, 0.1952252, -0.1483159, -0.1325612, 0.2789306, -0.4918891, -0.3207458, -0.4002184
    -0.0338265, 0.1094933, 0.1113708, -0.4262041, 0.3130188, 0.3035454, 0.0539090, -0.1708504
    0.2249388, 0.1499332, 0.0918251, -0.4048955, 0.2417646, -0.0781375, 0.0647991, 0.4362369
    -0.0282895, -0.0900536, -0.3221562, 0.0231988, -0.3404152, -0.0513410, -0.4174731, 0.0308473
    0.1668424, 0.3344521, -0.0532870, -0.0600087, 0.2670549, -0.0934474, -0.4218042, 0.1923514
    -0.4889445, 0.2732415, -0.2595133, -0.2856056, -0.2474788, -0.1976544, 0.3757972, -0.0276540
    -0.4311794, 0.0838393, -0.1905368, -0.2545608, 0.1115343, 0.0329114, 0.0388535, 0.1491540
    -0.2002401, -0.2041063, -0.3137326, -0.0346957, 0.2966585, 0.4597444, 0.1010034, 0.3098046
    -0.1656356, -0.0019984, -0.0007584, -0.1523754, -0.5199784, 0.3194352, -0.2137670, 0.1058149
    0.2952441, -0.2931790, 0.4705646, 0.0790619, 0.0003144, 0.1361744, -0.0528566, -0.1673936
    0.1318583, -0.0905288, -0.1440885, -0.2584444, -0.7371563, -0.4877339, -0.5890380, -0.3376481
    0.0799100, 0.3715304, 0.3661357, 0.5920555, 0.0229421, -0.0443000, -0.5298731, 0.3996252
    -0.3216403, 0.1283986, 0.0601108, 0.2566249, 0.1529905, -0.1653751, 0.2862226, 0.4111322
    -0.2634737, 0.3915212, 0.4506666, -0.1679726, -0.1495703, 0.0432177, -0.0700857, -0.3946955
    0.0720215, -0.1168483, 0.1301958, 0.0663297, 0.0076022, -0.1320583, -0.0072684, 0.0526766
    0.4005312, -0.0031333, -0.1216732, 0.2339514, 0.1652348, -0.1338500, 0.4973953, 0.3684065
    -0.4143495, 0.1780665, -0.0697868, -0.0997232, 0.0687763, -0.1456123, -0.2092715, 0.0189691
    -0.6826727, -0.6629136, -0.6555285, 0.3192035, -0.0694342, 0.2663665, -0.3917146, 0.0902561
    -0.5133109, -0.0766477, 0.0767347, -0.2457596, 0.1014029, -0.2873877, 0.0040285, 0.2393062
    0.0166857, 0.0309617, -0.1767922, -0.2731738, -0.1745891, 0.1539803, 0.2025868, 0.1977281
    -0.1848221, 0.0992378, -0.1108686, -0.1738138, -0.5793498, -0.3609751, -0.5280058, -0.0179569
    -0.4062726, -0.2277970, -0.2703095, -0.0866747, -0.4978129, -0.0251947, -0.0085684, 0.0232853
    0.0398995, -0.2167165, -0.0791776, 0.2240114, 0.1842670, -0.6018211, 0.1106252, -0.1592507
    -0.1362624, 0.2905875, -0.0013422, 0.0975723, -0.2237402, 0.0909775, -0.1894262, -0.1083135
    0.0, 0.0, 0.0, 0.0, 0.0, 0.0, 0.0, 0.0
    0.0, 0.0, 0.0, 0.0, 0.0, 0.0, 0.0, 0.0];

   // BsplineLUT 'l1_bspline': grid(15 pts) + table(4×16×15)
   w3 : ARRAY[0..14] OF REAL :=
[-3.0000000, -2.5714286, -2.1428571, -1.7142857, -1.2857143, -0.8571429, -0.4285714, 0.0
    0.4285714, 0.8571429, 1.2857143, 1.7142857, 2.1428571, 2.5714286, 3.0000000];
   w4 : ARRAY[0..959] OF REAL :=
[-0.1394233, -0.1411809, -0.1429312, -0.1446730, -0.1464052, -0.1481269, -0.1498369, -0.1515340
    -0.1532173, -0.1548856, -0.1565377, -0.1581727, -0.1597895, -0.1613868, -0.1629638, -0.0794552
    -0.0816418, -0.0837388, -0.0857477, -0.0876698, -0.0895068, -0.0912601, -0.0929311, -0.0945213
    -0.0960322, -0.0974653, -0.0988220, -0.1001038, -0.1013122, -0.1024486, -0.1252455, -0.1255447
    -0.1258071, -0.1260332, -0.1262234, -0.1263781, -0.1264976, -0.1265825, -0.1266330, -0.1266496
    -0.1266327, -0.1265826, -0.1264998, -0.1263847, -0.1262377, -0.0799751, -0.0787409, -0.0774544
    -0.0761172, -0.0747307, -0.0732965, -0.0718162, -0.0702913, -0.0687232, -0.0671136, -0.0654639
    -0.0637757, -0.0620505, -0.0602898, -0.0584952, -0.1070225, -0.1088643, -0.1106777, -0.1124617
    -0.1142155, -0.1159381, -0.1176288, -0.1192864, -0.1209103, -0.1224994, -0.1240529, -0.1255698
    -0.1270494, -0.1284905, -0.1298924, 0.0177095, 0.0175483, 0.0174157, 0.0173108, 0.0172329
    0.0171813, 0.0171551, 0.0171537, 0.0171762, 0.0172218, 0.0172899, 0.0173797, 0.0174903
    0.0176211, 0.0177712, -0.0182075, -0.0185586, -0.0189078, -0.0192552, -0.0196007, -0.0199444
    -0.0202862, -0.0206262, -0.0209644, -0.0213007, -0.0216351, -0.0219677, -0.0222984, -0.0226272
    -0.0229542, 0.0624644, 0.0627378, 0.0630123, 0.0632867, 0.0635600, 0.0638311, 0.0640990
    0.0643625, 0.0646206, 0.0648721, 0.0651160, 0.0653513, 0.0655768, 0.0657915, 0.0659942
    0.0749737, 0.0754191, 0.0757671, 0.0760200, 0.0761801, 0.0762498, 0.0762315, 0.0761274
    0.0759400, 0.0756716, 0.0753245, 0.0749010, 0.0744036, 0.0738345, 0.0731961, -0.1588649
    -0.1594506, -0.1599677, -0.1604175, -0.1608008, -0.1611191, -0.1613732, -0.1615644, -0.1616936
    -0.1617621, -0.1617709, -0.1617211, -0.1616139, -0.1614503, -0.1612314, 0.1175059, 0.1171356
    0.1166575, 0.1160742, 0.1153883, 0.1146024, 0.1137192, 0.1127412, 0.1116710, 0.1105112
    0.1092644, 0.1079333, 0.1065204, 0.1050283, 0.1034597, 0.0420621, 0.0404982, 0.0389136
    0.0373104, 0.0356906, 0.0340564, 0.0324097, 0.0307528, 0.0290877, 0.0274165, 0.0257413
    0.0240641, 0.0223871, 0.0207123, 0.0190418, 0.0036802, 0.0030620, 0.0024709, 0.0019069
    0.0013699, 0.0008601, 0.0003773, -0.0000785, -0.0005071, -0.0009088, -0.0012833, -0.0016308
    -0.0019512, -0.0022446, -0.0025110, -0.0811079, -0.0792010, -0.0773131, -0.0754445, -0.0735953
    -0.0717658, -0.0699560, -0.0681661, -0.0663965, -0.0646471, -0.0629183, -0.0612103, -0.0595231
    -0.0578570, -0.0562121, 0.1101897, 0.1101652, 0.1100717, 0.1099112, 0.1096858, 0.1093976
    0.1090486, 0.1086409, 0.1081766, 0.1076576, 0.1070862, 0.1064643, 0.1057939, 0.1050773
    0.1043164, 0.1828256, 0.1837029, 0.1844654, 0.1851155, 0.1856555, 0.1860879, 0.1864147
    0.1866386, 0.1867617, 0.1867865, 0.1867152, 0.1865502, 0.1862939, 0.1859487, 0.1855167
    0.0595048, 0.0615242, 0.0634741, 0.0653550, 0.0671674, 0.0689119, 0.0705890, 0.0721993
    0.0737432, 0.0752214, 0.0766343, 0.0779825, 0.0792665, 0.0804868, 0.0816440, 0.0235539
    0.0235894, 0.0235977, 0.0235797, 0.0235368, 0.0234700, 0.0233804, 0.0232693, 0.0231377
    0.0229868, 0.0228178, 0.0226317, 0.0224297, 0.0222131, 0.0219828, 0.0478683, 0.0472543
    0.0466411, 0.0460280, 0.0454145, 0.0448002, 0.0441846, 0.0435671, 0.0429473, 0.0423247
    0.0416988, 0.0410691, 0.0404351, 0.0397963, 0.0391521, 0.0072556, 0.0085569, 0.0098592
    0.0111617, 0.0124637, 0.0137644, 0.0150629, 0.0163584, 0.0176501, 0.0189372, 0.0202189
    0.0214944, 0.0227629, 0.0240236, 0.0252756, -0.1190253, -0.1196260, -0.1201990, -0.1207443
    -0.1212616, -0.1217509, -0.1222120, -0.1226448, -0.1230492, -0.1234252, -0.1237724, -0.1240908
    -0.1243804, -0.1246409, -0.1248722, 0.1018610, 0.1029626, 0.1040318, 0.1050682, 0.1060713
    0.1070410, 0.1079766, 0.1088780, 0.1097446, 0.1105761, 0.1113721, 0.1121322, 0.1128561
    0.1135433, 0.1141935, -0.0705152, -0.0710657, -0.0716057, -0.0721345, -0.0726515, -0.0731559
    -0.0736471, -0.0741245, -0.0745874, -0.0750351, -0.0754670, -0.0758824, -0.0762807, -0.0766611
    -0.0770231, -0.0909490, -0.0913742, -0.0917407, -0.0920498, -0.0923029, -0.0925011, -0.0926457
    -0.0927379, -0.0927792, -0.0927706, -0.0927134, -0.0926090, -0.0924585, -0.0922633, -0.0920245
    0.1135822, 0.1134194, 0.1132657, 0.1131207, 0.1129842, 0.1128561, 0.1127359, 0.1126236
    0.1125188, 0.1124212, 0.1123307, 0.1122469, 0.1121697, 0.1120987, 0.1120338, 0.0892454
    0.0891656, 0.0890862, 0.0890062, 0.0889244, 0.0888399, 0.0887515, 0.0886583, 0.0885591
    0.0884530, 0.0883389, 0.0882156, 0.0880823, 0.0879377, 0.0877809, -0.0596774, -0.0614152
    -0.0631330, -0.0648300, -0.0665055, -0.0681587, -0.0697888, -0.0713950, -0.0729764, -0.0745324
    -0.0760621, -0.0775647, -0.0790395, -0.0804856, -0.0819023, 0.0665300, 0.0666164, 0.0666485
    0.0666276, 0.0665551, 0.0664324, 0.0662605, 0.0660411, 0.0657752, 0.0654642, 0.0651095
    0.0647124, 0.0642740, 0.0637959, 0.0632792, -0.1160357, -0.1159643, -0.1158672, -0.1157443
    -0.1155953, -0.1154200, -0.1152182, -0.1149897, -0.1147341, -0.1144514, -0.1141413, -0.1138035
    -0.1134378, -0.1130441, -0.1126221, 0.0199476, 0.0177244, 0.0154825, 0.0132232, 0.0109476
    0.0086569, 0.0063521, 0.0040345, 0.0017051, -0.0006348, -0.0029843, -0.0053420, -0.0077069
    -0.0100779, -0.0124538, -0.0589397, -0.0581607, -0.0572549, -0.0562258, -0.0550771, -0.0538124
    -0.0524353, -0.0509494, -0.0493584, -0.0476659, -0.0458755, -0.0439909, -0.0420156, -0.0399532
    -0.0378075, -0.0787482, -0.0789619, -0.0791664, -0.0793615, -0.0795466, -0.0797217, -0.0798863
    -0.0800402, -0.0801831, -0.0803146, -0.0804345, -0.0805424, -0.0806381, -0.0807212, -0.0807914
    -0.0659224, -0.0641469, -0.0623249, -0.0604586, -0.0585500, -0.0566012, -0.0546145, -0.0525918
    -0.0505353, -0.0484471, -0.0463294, -0.0441842, -0.0420137, -0.0398200, -0.0376051, 0.0625157
    0.0632284, 0.0639766, 0.0647592, 0.0655750, 0.0664229, 0.0673015, 0.0682097, 0.0691464
    0.0701102, 0.0711001, 0.0721149, 0.0731532, 0.0742140, 0.0752961, 0.0149698, 0.0139133
    0.0128017, 0.0116372, 0.0104224, 0.0091595, 0.0078510, 0.0064992, 0.0051066, 0.0036755
    0.0022083, 0.0007074, -0.0008249, -0.0023860, -0.0039738, 0.0290725, 0.0282233, 0.0273817
    0.0265474, 0.0257202, 0.0248999, 0.0240864, 0.0232795, 0.0224789, 0.0216846, 0.0208962
    0.0201136, 0.0193367, 0.0185652, 0.0177989, 0.0344971, 0.0378870, 0.0412622, 0.0446213
    0.0479634, 0.0512872, 0.0545917, 0.0578756, 0.0611378, 0.0643773, 0.0675927, 0.0707831
    0.0739473, 0.0770841, 0.0801924, -0.0421340, -0.0431118, -0.0440828, -0.0450455, -0.0459982
    -0.0469394, -0.0478675, -0.0487809, -0.0496780, -0.0505573, -0.0514172, -0.0522560, -0.0530723
    -0.0538643, -0.0546307, -0.1622524, -0.1621790, -0.1620038, -0.1617292, -0.1613578, -0.1608921
    -0.1603347, -0.1596880, -0.1589546, -0.1581371, -0.1572378, -0.1562594, -0.1552044, -0.1540753
    -0.1528746, -0.0090858, -0.0075867, -0.0061187, -0.0046829, -0.0032802, -0.0019117, -0.0005783
    0.0007190, 0.0019792, 0.0032014, 0.0043844, 0.0055274, 0.0066293, 0.0076891, 0.0087060
    0.0064042, 0.0070511, 0.0076863, 0.0083093, 0.0089194, 0.0095160, 0.0100985, 0.0106663
    0.0112187, 0.0117551, 0.0122749, 0.0127776, 0.0132623, 0.0137287, 0.0141759, -0.0177168
    -0.0166479, -0.0155266, -0.0143542, -0.0131325, -0.0118628, -0.0105469, -0.0091862, -0.0077823
    -0.0063367, -0.0048511, -0.0033270, -0.0017659, -0.0001694, 0.0014610, -0.0314599, -0.0320327
    -0.0326800, -0.0333999, -0.0341903, -0.0350491, -0.0359744, -0.0369640, -0.0380159, -0.0391281
    -0.0402986, -0.0415253, -0.0428061, -0.0441390, -0.0455221, 0.0591273, 0.0582139, 0.0572240
    0.0561600, 0.0550244, 0.0538195, 0.0525478, 0.0512118, 0.0498138, 0.0483565, 0.0468421
    0.0452731, 0.0436521, 0.0419813, 0.0402634, -0.0462357, -0.0461251, -0.0460184, -0.0459164
    -0.0458196, -0.0457286, -0.0456441, -0.0455667, -0.0454970, -0.0454356, -0.0453832, -0.0453403
    -0.0453077, -0.0452858, -0.0452754, -0.0598098, -0.0618588, -0.0639245, -0.0660049, -0.0680977
    -0.0702008, -0.0723122, -0.0744296, -0.0765509, -0.0786741, -0.0807969, -0.0829172, -0.0850329
    -0.0871419, -0.0892420, 0.0654971, 0.0660617, 0.0665634, 0.0670037, 0.0673837, 0.0677048
    0.0679682, 0.0681753, 0.0683272, 0.0684253, 0.0684709, 0.0684652, 0.0684095, 0.0683051
    0.0681533, -0.0077130, -0.0083153, -0.0089273, -0.0095481, -0.0101767, -0.0108123, -0.0114539
    -0.0121007, -0.0127516, -0.0134059, -0.0140625, -0.0147206, -0.0153793, -0.0160376, -0.0166946
    -0.0487178, -0.0471633, -0.0456145, -0.0440716, -0.0425349, -0.0410044, -0.0394806, -0.0379635
    -0.0364535, -0.0349506, -0.0334552, -0.0319675, -0.0304876, -0.0290159, -0.0275525, -0.0120348
    -0.0133224, -0.0146009, -0.0158700, -0.0171297, -0.0183796, -0.0196196, -0.0208496, -0.0220692
    -0.0232784, -0.0244769, -0.0256645, -0.0268410, -0.0280063, -0.0291601, 0.1104566, 0.1098977
    0.1092816, 0.1086091, 0.1078807, 0.1070971, 0.1062589, 0.1053668, 0.1044213, 0.1034232
    0.1023731, 0.1012716, 0.1001194, 0.0989171, 0.0976653, -0.0693738, -0.0700046, -0.0705503
    -0.0710135, -0.0713968, -0.0717027, -0.0719339, -0.0720929, -0.0721823, -0.0722047, -0.0721627
    -0.0720588, -0.0718957, -0.0716760, -0.0714021, 0.0144107, 0.0149072, 0.0154286, 0.0159744
    0.0165441, 0.0171373, 0.0177535, 0.0183921, 0.0190528, 0.0197350, 0.0204382, 0.0211620
    0.0219059, 0.0226693, 0.0234519, -0.0856846, -0.0857019, -0.0856579, -0.0855545, -0.0853933
    -0.0851765, -0.0849057, -0.0845828, -0.0842096, -0.0837880, -0.0833199, -0.0828070, -0.0822512
    -0.0816544, -0.0810183, 0.1129993, 0.1151353, 0.1173310, 0.1195833, 0.1218886, 0.1242438
    0.1266453, 0.1290900, 0.1315744, 0.1340952, 0.1366491, 0.1392326, 0.1418425, 0.1444754
    0.1471280, 0.1679913, 0.1680896, 0.1680988, 0.1680210, 0.1678583, 0.1676128, 0.1672865
    0.1668818, 0.1664005, 0.1658449, 0.1652170, 0.1645190, 0.1637529, 0.1629209, 0.1620251
    -0.1020884, -0.1013920, -0.1006600, -0.0998936, -0.0990941, -0.0982626, -0.0974004, -0.0965087
    -0.0955887, -0.0946415, -0.0936685, -0.0926709, -0.0916498, -0.0906064, -0.0895421, -0.0705225
    -0.0704993, -0.0704878, -0.0704866, -0.0704946, -0.0705105, -0.0705332, -0.0705614, -0.0705940
    -0.0706298, -0.0706674, -0.0707058, -0.0707437, -0.0707799, -0.0708131, -0.1320913, -0.1321882
    -0.1322562, -0.1322947, -0.1323030, -0.1322805, -0.1322265, -0.1321404, -0.1320215, -0.1318692
    -0.1316827, -0.1314614, -0.1312048, -0.1309121, -0.1305827, -0.1371553, -0.1334958, -0.1297319
    -0.1258684, -0.1219103, -0.1178626, -0.1137300, -0.1095175, -0.1052300, -0.1008724, -0.0964495
    -0.0919664, -0.0874279, -0.0828388, -0.0782042, 0.0085733, 0.0085398, 0.0084969, 0.0084456
    0.0083870, 0.0083219, 0.0082513, 0.0081763, 0.0080979, 0.0080170, 0.0079346, 0.0078516
    0.0077692, 0.0076882, 0.0076097, 0.0226030, 0.0203749, 0.0180662, 0.0156800, 0.0132194
    0.0106876, 0.0080877, 0.0054228, 0.0026960, -0.0000894, -0.0029303, -0.0058237, -0.0087663
    -0.0117551, -0.0147868, -0.1211590, -0.1201795, -0.1191991, -0.1182173, -0.1172332, -0.1162465
    -0.1152565, -0.1142624, -0.1132637, -0.1122599, -0.1112502, -0.1102340, -0.1092108, -0.1081799
    -0.1071406, -0.0816189, -0.0836604, -0.0856507, -0.0875902, -0.0894792, -0.0913182, -0.0931074
    -0.0948471, -0.0965379, -0.0981799, -0.0997735, -0.1013191, -0.1028170, -0.1042675, -0.1056711];

   // MatMul 'l1_base': W(4×16) + b(4)
   w5 : ARRAY[0..67] OF REAL :=
[-0.2824876, -0.6565906, -0.3122313, 0.3330409, -0.2412571, -0.1209215, -0.1549156, 0.0219229
    -0.7318159, -0.3782304, 0.1660175, -0.4863215, 0.1786766, 0.1779261, 0.1966676, 0.0488548
    0.0575393, 0.3588348, -0.1176801, 0.2243771, 0.0563377, 0.3474633, 0.2406189, -0.3899010
    -0.1843529, 0.2943886, -0.3224228, -0.3371529, -0.3695943, -0.0532869, -0.5337853, -0.5914542
    0.1487857, 0.1035332, -0.1314158, -0.2367104, 0.3866917, -0.0002227, -0.2907901, -0.0284536
    0.2614560, 0.0448420, 0.3463572, 0.3907122, 0.3632395, -0.4534223, 0.4758949, 0.0794281
    0.3638572, -0.2039453, 0.4670161, -0.1860616, -0.3569592, -0.4310024, 0.2556136, 0.3338891
    0.2300281, -0.0679060, -0.3959090, -0.1938804, 0.3476668, 0.1242622, -0.3246959, -0.0931496
    0.0, 0.0, 0.0, 0.0];

   // Total: 6 array blocks
   END_STRUCT;
BEGIN
END_DATA_BLOCK

FUNCTION "BsplineEval" : REAL
{ S7_Optimized_Access := 'FALSE' }
VERSION : 0.1
VAR_INPUT
    x : REAL;
    lut_grid : ARRAY[0..14] OF REAL;
    lut_table : ARRAY[0..14] OF REAL;
END_VAR
VAR_TEMP
    lo, hi, mid : INT;
    t, vlo, vhi : REAL;
END_VAR

BEGIN
    // Binary search for interval containing x
    lo := 0;
    hi := 14;
    WHILE hi - lo > 1 DO
        mid := lo + (hi - lo) / 2;
        IF x > lut_grid[mid] THEN lo := mid; ELSE hi := mid; END_IF;
    END_WHILE;

    // Linear interpolation: y = vlo*(1-t) + vhi*t
    vlo := lut_table[lo];
    vhi := lut_table[hi];
    t := (x - lut_grid[lo]) / (lut_grid[hi] - lut_grid[lo] + 1.0E-10);
    "BsplineEval" := vlo * (1.0 - t) + vhi * t;
END_FUNCTION

FUNCTION_BLOCK "NeuroPLC_Inference"
{ S7_Optimized_Access := 'FALSE' }
VERSION : 0.1
VAR_INPUT
    features : ARRAY[0..27] OF REAL;
END_VAR

VAR_OUTPUT
    fault_class : INT;
    confidence : REAL;
END_VAR

VAR
    i, j, k : INT;
    sum_val, max_val, t_val : REAL;
    v0 : ARRAY[0..27] OF REAL;
    v1 : ARRAY[0..27] OF REAL;
    v3 : ARRAY[0..15, 0..27] OF REAL;
    v2 : ARRAY[0..15] OF REAL;
    v4 : ARRAY[0..15] OF REAL;
    v5 : ARRAY[0..15] OF REAL;
    v7 : ARRAY[0..3, 0..15] OF REAL;
    v6 : ARRAY[0..3] OF REAL;
    v8 : ARRAY[0..3] OF REAL;
    v9 : ARRAY[0..3] OF REAL;
    lut_tmp : ARRAY[0..14] OF REAL;
END_VAR

BEGIN
    // ---- Input ----
    FOR i := 0 TO 27 DO
        v0[i] := features[i];
    END_FOR;

    // ---- l0_silu: SILU ----
    v1[0] := v0[0] / (1.0 + EXP(-v0[0]));
    v1[1] := v0[1] / (1.0 + EXP(-v0[1]));
    v1[2] := v0[2] / (1.0 + EXP(-v0[2]));
    v1[3] := v0[3] / (1.0 + EXP(-v0[3]));
    v1[4] := v0[4] / (1.0 + EXP(-v0[4]));
    v1[5] := v0[5] / (1.0 + EXP(-v0[5]));
    v1[6] := v0[6] / (1.0 + EXP(-v0[6]));
    v1[7] := v0[7] / (1.0 + EXP(-v0[7]));
    v1[8] := v0[8] / (1.0 + EXP(-v0[8]));
    v1[9] := v0[9] / (1.0 + EXP(-v0[9]));
    v1[10] := v0[10] / (1.0 + EXP(-v0[10]));
    v1[11] := v0[11] / (1.0 + EXP(-v0[11]));
    v1[12] := v0[12] / (1.0 + EXP(-v0[12]));
    v1[13] := v0[13] / (1.0 + EXP(-v0[13]));
    v1[14] := v0[14] / (1.0 + EXP(-v0[14]));
    v1[15] := v0[15] / (1.0 + EXP(-v0[15]));
    v1[16] := v0[16] / (1.0 + EXP(-v0[16]));
    v1[17] := v0[17] / (1.0 + EXP(-v0[17]));
    v1[18] := v0[18] / (1.0 + EXP(-v0[18]));
    v1[19] := v0[19] / (1.0 + EXP(-v0[19]));
    v1[20] := v0[20] / (1.0 + EXP(-v0[20]));
    v1[21] := v0[21] / (1.0 + EXP(-v0[21]));
    v1[22] := v0[22] / (1.0 + EXP(-v0[22]));
    v1[23] := v0[23] / (1.0 + EXP(-v0[23]));
    v1[24] := v0[24] / (1.0 + EXP(-v0[24]));
    v1[25] := v0[25] / (1.0 + EXP(-v0[25]));
    v1[26] := v0[26] / (1.0 + EXP(-v0[26]));
    v1[27] := v0[27] / (1.0 + EXP(-v0[27]));

